// TwinCAT 3 PLC project StudentStation
// ProgramVersion: 3.1.4022.4
// libraries:
//   Tc2_Standard, * (Beckhoff Automation GmbH)
//   Tc2_System, * (Beckhoff Automation GmbH)
//   Tc3_Module, * (Beckhoff Automation GmbH)
//   VisuDialogs, * (System)
//   VisuSymbols,3.5.10.0,System
// project tree:
//   ABBControl/ ABBAssemble.TcPOU, ABBGotoAGVPos.TcPOU, ABBGotoBuffer.TcPOU, ABBGotoHome.TcPOU, ABBGotoScanner.TcPOU, ABBGotoTable.TcPOU, ABBPickLeaveBuffer.TcPOU, ABBPickLeaveContainerAGV.TcPOU, ABBPickLeaveContaineronTable.TcPOU, ABBPickLeaveScanner.TcPOU, ABBScanContainer.TcPOU, ABBScannerStation.TcPOU
//   Automation Library/ AGVControlSystem.TcPOU, AutomationLibrary.TcPOU, BookingSystem.TcPOU, CommData.TcGVL, OrderHandling.TcPOU, PhysicalSystemTest.TcPOU, RobotControlSystem.TcPOU, RobotPosTracker.TcPOU, SensorReader.TcPOU, Visualaisation_Control.TcPOU
//   DUTs/ ABBPositions.TcDUT, ABBXYPOS.TcDUT, OrderPLC.TcDUT, PLCRobotOrder.TcDUT, Station.TcDUT, Storage.TcDUT
//   / GlobalTextList.TcGTLO, PlcTask.TcTTO, Visualization Manager.TcVMO (not stored)
//   GVLs/ GVL.TcGVL
//   POUs/ ABB_Control_FB.TcPOU, MAIN.TcPOU, Scanner_FB.TcPOU, Sensor_Sense.TcPOU
//   VISUs/ RobotStation.TcVIS, Station.TcVIS, Visualization.TcVIS
// real-time tasks:
//   TASK PlcTask: cycle T#10ms, priority 20, ADS port 350

CONFIGURATION StudentStation
    RESOURCE PLC ON TwinCAT3
        TASK PlcTask(INTERVAL := T#10ms, PRIORITY := 20);
        PROGRAM MAIN WITH PlcTask : MAIN;
    END_RESOURCE
END_CONFIGURATION

// ---- DUTs/ABBPositions.TcDUT
TYPE ABBPositions :
STRUCT
	Home: ABBXYPOS;
	Bufferhome: ABBXYPOS;
	Scannerhome: ABBXYPOS;
	Tablehome: ABBXYPOS;
	AGVPOShome: ABBXYPOS;
	Storage1: ABBXYPOS;
	Storage2: ABBXYPOS;
	Storage3: ABBXYPOS;
END_STRUCT
END_TYPE

// ---- DUTs/ABBXYPOS.TcDUT
TYPE ABBXYPOS :
STRUCT
	X:	INT;
	Y:	INT;
END_STRUCT
END_TYPE

// ---- DUTs/OrderPLC.TcDUT
TYPE OrderPLC :
STRUCT
	RobotPOS:STRING; //Prerequest position for the robot to do the step
	PLCorder:INT;	//PLCStep Code
	Robotreply:INT;	//Robot Response Code
END_STRUCT
END_TYPE

// ---- DUTs/PLCRobotOrder.TcDUT
TYPE PLCRobotOrder :
STRUCT
	GotoHome: OrderPLC;
	GotoAGVPos: OrderPLC;
	GotoBuffer: OrderPLC;
	GotoScanner: OrderPLC;
	GotoTable: OrderPLC;
END_STRUCT
END_TYPE

// ---- DUTs/Station.TcDUT
TYPE Station :
STRUCT
	Storage1: Storage;
	Storage2: Storage;
	Storage3: Storage;
END_STRUCT
END_TYPE

// ---- DUTs/Storage.TcDUT
TYPE Storage :
STRUCT
	Component: STRING;
	Quatity: INT;
END_STRUCT
END_TYPE

// ---- Automation Library/CommData.TcGVL
{attribute 'qualified_only'}
VAR_GLOBAL
	msProductNames : ARRAY[1..9] OF STRING := ['BLUECYLINDER', 'BLUEOCTAGON', 'BLUEPLATE', 'YELLOWCYLINDER', 'YELLOWOCTAGON', 'YELLOWPLATE', 'REDCYLINDER', 'REDOCTAGON', 'REDPLATE'];
	mxRequestAGV: BOOL;
	mxAGVOutsideStation: BOOL;
	mxAGVLeaveStation: BOOL;
	mwAGVinStationPOS: INT := -700;
	mwAGVinOutsidePOS: INT := 0;
	mwCurrentAGVPOS: INT;
	ABBPostions: ABBPositions := (Bufferhome := (X := -185, Y := 250), Scannerhome := (X := -185, Y := 180), Tablehome := (X := -185, Y :=350), AGVPOShome := (X := -60, Y := 350), Storage1 := (X := -315, Y := 180), Storage2 := (X := -315, Y := 350), Storage3 := (X := -60, Y := 180));
	mxOnlineMode: BOOL;
	mxABBExecuting: BOOL;
	mwXaxis: INT;
	mwYaxis: INT;
	mxGripper: BOOL;
	mwABBPosXaxis: INT;
	mwABBPosYaxis: INT;
	mxStartABB: BOOL;
	mxScannernoobject:BOOL;
	mxWaitingforSensorinput:BOOL;
	mxNewBookingrequest: BOOL;
	
	
	//Robot Control Signals
	mxRobotOnline AT %I*:BOOL;
	msRobotLastPos:STRING;
	qwOrderRobot AT %Q*:DINT;
	iwReplyRobot AT %I*:DINT;
	qxPLCStrobe AT %Q*:BOOL;
	ixRobotStrobe AT %I*:BOOL;
	iwProgressRobot AT %I*: INT;
	maOrderMaker: ARRAY[1..6] OF INT;
END_VAR

// ---- GVLs/GVL.TcGVL
{attribute 'qualified_only'}
VAR_GLOBAL
	// Order for the next assembly part. The part name should be sent as per the part list and case sensitive. 
	{attribute 'OPC.UA.DA' := '1'}
	qsOrderFornextAssembly AT %Q*: STRING := '0';
	// Parts in your Station buffer. Each buffer have 3 storage locations. The part name and quantity should be mentioned.
	{attribute 'OPC.UA.DA' := '1'}
	BufferProducts AT %Q*: Station;
	// Signal to AGV, a pallet is placed from Station to the AGV. 
	{attribute 'OPC.UA.DA' := '1'}
	qxPalletPlacedinAGV AT %Q*: BOOL;
	// Signal From AGV, that it have docked in your station
	{attribute 'OPC.UA.DA' := '1'}
	ixAGVatStation AT %I*: BOOL;
	{attribute 'OPC.UA.DA' := '1'}	
	qxPickedfromAGV AT %Q*:BOOL; //Part is picked up from the AGV
	{attribute 'OPC.UA.DA' := '1'}
	mwStationStatus AT %Q*: INT; //Pre-Conditioning Mode //100:Ready to Work § 200: Getting Booked § 300: Booked and Busy § 400 : Manual mode  § 500: Pause Mode § 1000 : Emergency Mode 
	{attribute 'OPC.UA.DA' := '1'}	
	// Emergency Stop is active
	ixEmergencyStop AT %Q*:BOOL;
	
	// Inductive sensor reading. from scaning station
	ixInductiveSensor1 AT %I*:BOOL;
	// Inductive sensor reading. from scaning station
	ixInductiveSensor2 AT %I*:BOOL;
	// Inductive sensor reading. from scaning station
	ixInductiveSensor3 AT %I*:BOOL;
	// Inductive sensor reading. from scaning station
	ixInductiveSensor4 AT %I*:BOOL;
	// Inductive sensor reading. from the sensor in robot Tool
	ixInductiveSensorinTool AT %I*:BOOL;
	// Station ID of the station you are working with.
	{attribute 'OPC.UA.DA' := '1'}
	mwStationID AT %Q*: INT;
	
END_VAR

// ---- POUs/MAIN.TcPOU
PROGRAM MAIN
VAR	
END_VAR

VAR_INPUT
	qxABBonlineLamp : BOOL;
	qxABBExecutLamp : BOOL;
	qxABBErrorLamp : BOOL;
	qxPauseLamp : BOOL;
	qxEmergySTLamp : BOOL;
	ixPauseButt : BOOL;
	ixResetABB : BOOL;
	qxAutoMode : BOOL;
	qxManualMode : BOOL;
	ixAutoLamp : BOOL;
	ixManualLamp : BOOL;
	qxDoneContainerScan : BOOL;
	qxDoneBuffer1Scan : BOOL;
	qsContainer : STRING;
	qsTask : STRING;
	qsSubTask : STRING;
	mxPlateAvailable : BOOL;
	mxCylinderAvailable : BOOL;
	mxOctagonAvailable : BOOL;
	mwBufferID : INT;
	ixEmptyBuffer : BOOL;
	mwPartID : INT;
	sPartID : ARRAY [1..3] OF STRING:= ['Part 1', 'Part 2', 'Part 3'];
END_VAR

VAR_OUTPUT
	
END_VAR

AutomationLibrary();
Visualaisation_Control();
RobotPosTracker();
ABB_Control_FB();

END_PROGRAM

// ---- Automation Library/AutomationLibrary.TcPOU
PROGRAM AutomationLibrary
VAR
	OrderHandling_Global: OrderHandling;
	mxErrorCodeOrder: INT;
	AGVControlSystem_GLobal: AGVControlSystem;
	RobotControlSystem_Global: RobotControlSystem;
	ABBGotoHome_TEST: ABBGotoHome;
	mxEnable: BOOL;
	BookingSystem_Global: BookingSystem;
	mxBookingDone: BOOL;
	mxBookingError: BOOL;
END_VAR

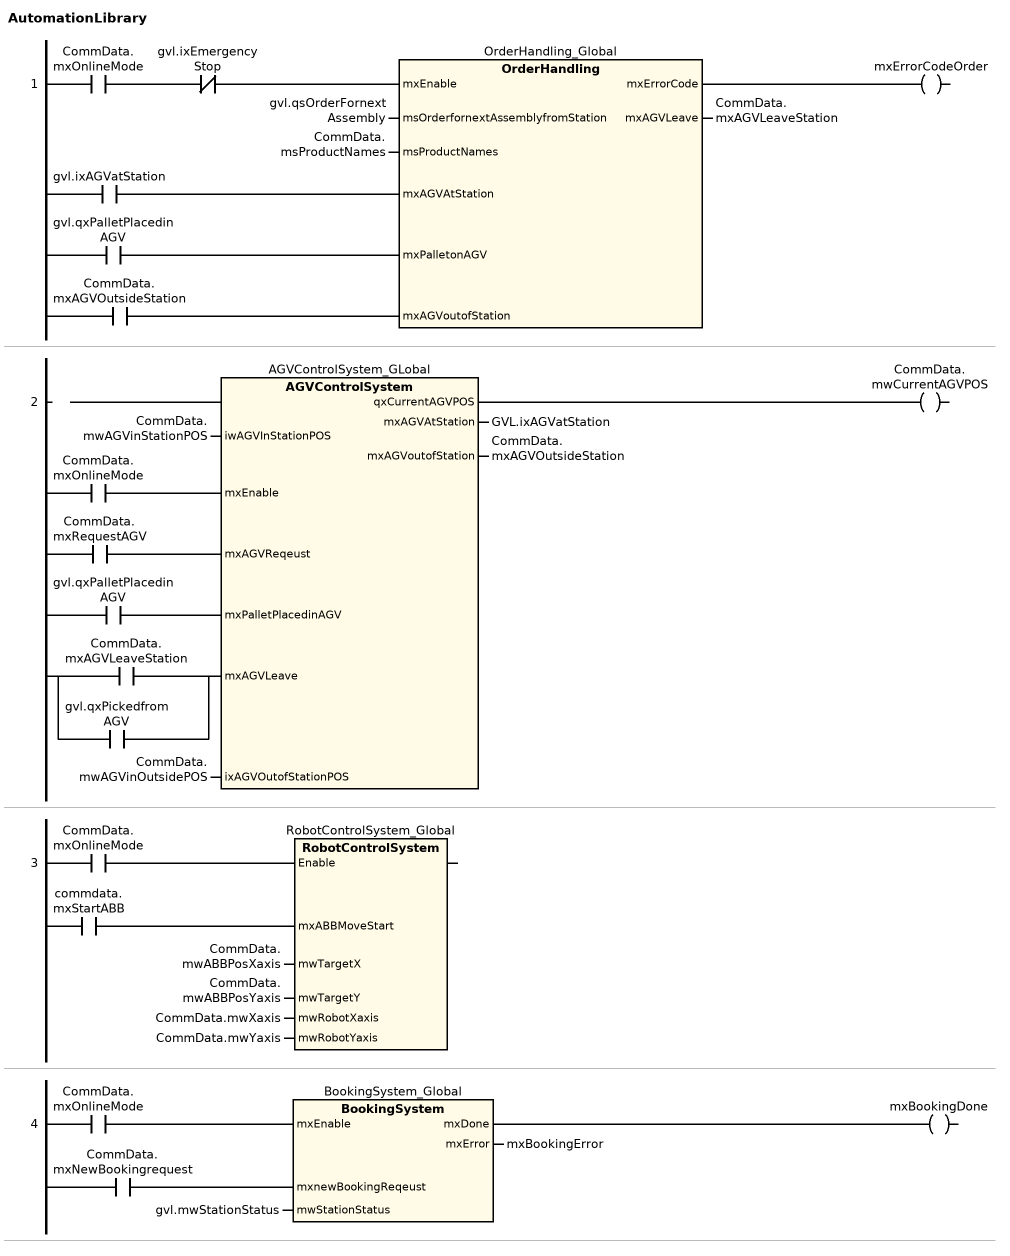
// NETWORK 1
OrderHandling_Global(
    mxEnable := CommData.mxOnlineMode AND NOT gvl.ixEmergencyStop,
    msOrderfornextAssemblyfromStation := gvl.qsOrderFornextAssembly,
    msProductNames := CommData.msProductNames,
    mxAGVAtStation := gvl.ixAGVatStation,
    mxPalletonAGV := gvl.qxPalletPlacedinAGV,
    mxAGVoutofStation := CommData.mxAGVOutsideStation,
    mxAGVLeave => CommData.mxAGVLeaveStation); // OrderHandling
mxErrorCodeOrder := OrderHandling_Global.mxErrorCode;

// NETWORK 2
AGVControlSystem_GLobal(
    iwAGVInStationPOS := CommData.mwAGVinStationPOS,
    mxEnable := CommData.mxOnlineMode,
    mxAGVReqeust := CommData.mxRequestAGV,
    mxPalletPlacedinAGV := gvl.qxPalletPlacedinAGV,
    mxAGVLeave := CommData.mxAGVLeaveStation OR gvl.qxPickedfromAGV,
    ixAGVOutofStationPOS := CommData.mwAGVinOutsidePOS,
    mxAGVAtStation => GVL.ixAGVatStation,
    mxAGVoutofStation => CommData.mxAGVOutsideStation); // AGVControlSystem
CommData.mwCurrentAGVPOS := AGVControlSystem_GLobal.qxCurrentAGVPOS;

// NETWORK 3
RobotControlSystem_Global(
    Enable := CommData.mxOnlineMode,
    mxABBMoveStart := commdata.mxStartABB,
    mwTargetX := CommData.mwABBPosXaxis,
    mwTargetY := CommData.mwABBPosYaxis,
    mwRobotXaxis := CommData.mwXaxis,
    mwRobotYaxis := CommData.mwYaxis); // RobotControlSystem

// NETWORK 4
BookingSystem_Global(
    mxEnable := CommData.mxOnlineMode,
    mxnewBookingReqeust := CommData.mxNewBookingrequest,
    mwStationStatus := gvl.mwStationStatus,
    mxError => mxBookingError); // BookingSystem
mxBookingDone := BookingSystem_Global.mxDone;

END_PROGRAM

// ---- Automation Library/OrderHandling.TcPOU
FUNCTION_BLOCK OrderHandling
VAR_INPUT
	mxEnable: BOOL;
	msOrderfornextAssemblyfromStation: STRING;
	msProductNames: Array[1..9] OF STRING;
	mxAGVAtStation: BOOL;
	mxPalletonAGV: BOOL;
	mxAGVoutofStation: BOOL;
END_VAR
VAR_OUTPUT
	mxErrorCode: INT;
	mxAGVLeave: BOOL;
END_VAR
VAR
	order: INT;
END_VAR

IF mxEnable THEN
	CASE order OF
		0:
			IF msOrderfornextAssemblyfromStation <> '0' THEN
				order:= 10;
			END_IF
		10:
			order:=20;
		20:
			IF msOrderfornextAssemblyfromStation = msProductNames[1] THEN
				order:=30;
			ELSIF msOrderfornextAssemblyfromStation = msProductNames[2] THEN
				order:=30;
			ELSIF msOrderfornextAssemblyfromStation = msProductNames[3] THEN
				order:=30;
			ELSIF msOrderfornextAssemblyfromStation = msProductNames[4] THEN
				order:=30;
			ELSIF msOrderfornextAssemblyfromStation = msProductNames[5] THEN
				order:=30;
			ELSIF msOrderfornextAssemblyfromStation = msProductNames[6] THEN
				order:=30;
			ELSIF msOrderfornextAssemblyfromStation = msProductNames[7] THEN
				order:=30;
			ELSIF msOrderfornextAssemblyfromStation = msProductNames[8] THEN
				order:=30;
			ELSIF msOrderfornextAssemblyfromStation = msProductNames[9] THEN
				order:=30;
			ELSIF msOrderfornextAssemblyfromStation = 'AssembledProduct' THEN
				order:=30;
			ELSIF msOrderfornextAssemblyfromStation = 'InvalidPart' THEN
				order:=30;
			ELSE 
				order:=22;
			END_IF 
		22: // Invalid Product Name
			mxErrorCode:=22;
				IF msOrderfornextAssemblyfromStation = '0' THEN
					mxErrorCode:=0;
					order:= 0;
				END_IF
		30:
			CommData.mxRequestAGV:=TRUE;
			IF mxAGVAtStation THEN
				CommData.mxRequestAGV:=FALSE;
				order:=40;
			END_IF
		40:
			IF mxPalletonAGV THEN
				mxAGVLeave:=TRUE;
				order:=50;
			END_IF
		50:
			IF mxAGVoutofStation THEN
				mxAGVLeave:=FALSE;
				order:=60;
			END_IF
		60:
			IF msOrderfornextAssemblyfromStation = '0' THEN
				order:= 0;
			END_IF
	END_CASE
END_IF

END_FUNCTION_BLOCK

// ---- Automation Library/AGVControlSystem.TcPOU
FUNCTION_BLOCK AGVControlSystem
VAR
	AGV: INT;
	mxAGVMoveTarget: INT;
	iwAGVOutofStationPOS: INT;
	RSpeed:INT:=1;
END_VAR
VAR_INPUT
	iwAGVInStationPOS: INT;
	mxEnable: BOOL;
END_VAR
VAR_OUTPUT
	qxCurrentAGVPOS: INT := 0;
	mxAGVAtStation: BOOL;
	mxAGVoutofStation: BOOL;
END_VAR
VAR_INPUT
	mxAGVReqeust: BOOL;
	mxPalletPlacedinAGV: BOOL;
	mxAGVLeave: BOOL;
	ixAGVOutofStationPOS: INT;
END_VAR

IF mxEnable THEN
	
	CASE AGV OF
		0:
			IF mxAGVReqeust THEN
				AGV:=10;
			END_IF
		10:
			mxAGVMoveTarget:= iwAGVInStationPOS;
			AGV:=20;
		20:
			
			IF mxAGVMoveTarget < qxCurrentAGVPOS THEN
				qxCurrentAGVPOS:=qxCurrentAGVPOS-RSpeed;
				AGV:=30;
			END_IF
		30:
			IF mxAGVMoveTarget < qxCurrentAGVPOS THEN
				AGV:=20;
			ELSIF  mxAGVMoveTarget >= qxCurrentAGVPOS THEN
				AGV:=40;
			END_IF
		40:
			mxAGVAtStation:=TRUE;
			IF mxPalletPlacedinAGV OR mxAGVLeave THEN
				mxAGVAtStation:=FALSE;
				AGV:=50;
			END_IF
		50:
			mxAGVMoveTarget:= iwAGVOutofStationPOS;
			AGV:=60;
		60:
			IF mxAGVMoveTarget > qxCurrentAGVPOS THEN
				qxCurrentAGVPOS:=qxCurrentAGVPOS+RSpeed;
				AGV:=70;
			END_IF
		70:
			IF mxAGVMoveTarget > qxCurrentAGVPOS THEN
				AGV:=60;
			ELSIF  mxAGVMoveTarget <= qxCurrentAGVPOS THEN
				AGV:=80;
			END_IF
		80:
			mxAGVoutofStation:=TRUE;
			IF NOT mxAGVReqeust AND NOT mxAGVLeave THEN
				mxAGVoutofStation:=FALSE;
				AGV:=0;
			END_IF
	END_CASE
		
END_IF

END_FUNCTION_BLOCK

// ---- Automation Library/RobotControlSystem.TcPOU
FUNCTION_BLOCK RobotControlSystem
VAR_INPUT
	Enable: BOOL;
	mxABBMoveStart: BOOL;
	mwTargetX: INT;
	mwTargetY: INT;
END_VAR
VAR_OUTPUT
END_VAR
VAR
	ABBMove: INT;
	RSpeed:INT:=1;
END_VAR

VAR_IN_OUT
	mwRobotXaxis: INT;
	mwRobotYaxis: INT;
END_VAR

IF Enable THEN
	CASE ABBMove OF
		0:
			IF mxABBMoveStart THEN
				ABBMove:=10;
			END_IF
		10:
			IF NOT CommData.mxABBExecuting THEN
				CommData.mxABBExecuting:=TRUE;
				ABBMove:=20;
			END_IF
		20:
			IF mwRobotXaxis < mwTargetX THEN
				mwRobotXaxis :=mwRobotXaxis+RSpeed;
				ABBMove:=30;
			ELSIF mwRobotXaxis > mwTargetX THEN
				mwRobotXaxis :=mwRobotXaxis-RSpeed;
				ABBMove:=30;
			ELSIF mwRobotXaxis = mwTargetX THEN
				ABBMove:=30;
			END_IF
		30:
			IF mwRobotYaxis < mwTargetY THEN
				mwRobotYaxis :=mwRobotYaxis+RSpeed;
				ABBMove:=40;
			ELSIF mwRobotYaxis > mwTargetY THEN
				mwRobotYaxis :=mwRobotYaxis-RSpeed;
				ABBMove:=40;
			ELSIF mwRobotYaxis = mwTargetY THEN
				ABBMove:=40;
			END_IF
		40:
			IF mwRobotXaxis = mwTargetX AND mwRobotYaxis = mwTargetY THEN
				ABBMove:=50;
			ELSIF gvl.ixEmergencyStop THEN
				ABBMove:=50;
			ELSE
				ABBMOve:=20;
			END_IF
		50:
			CommData.mxABBExecuting:=FALSE;
			IF NOT mxABBMoveStart THEN
				ABBMove:=0;
			END_IF
	END_CASE
END_IF

END_FUNCTION_BLOCK

// ---- ABBControl/ABBGotoHome.TcPOU
FUNCTION_BLOCK ABBGotoHome
VAR_INPUT
	mxEnable: BOOL;
END_VAR
VAR_OUTPUT
	mxDone:BOOL;
	mxExecuting: BOOL;
	mxError: BOOL;
END_VAR
VAR
	ABB: INT;
END_VAR

CASE ABB OF
	0:
		IF mxEnable AND NOT CommData.mxABBExecuting THEN
			ABB:=10;
		END_IF
	10:
		IF CommData.mxRobotOnline THEN
			ABB:=100;
			ELSE
			ABB:=200;
		END_IF
	100:
		mxExecuting:=TRUE;
		CommData.maOrderMaker[1] := 1;
		CommData.maOrderMaker[2] := 0;
		CommData.maOrderMaker[3] := 0;
		CommData.maOrderMaker[4] := 0;
		CommData.maOrderMaker[5] := 0;
		CommData.maOrderMaker[6] := 0;
		CommData.qwOrderRobot:=100000;
		ABB:=101;
	101:
		IF CommData.qwOrderRobot > 0 THEN
			CommData.qxPLCStrobe:=TRUE;
			ABB:=102;
		END_IF
	102:
		IF CommData.ixRobotStrobe THEN
			IF CommData.iwReplyRobot = CommData.qwOrderRobot+1 THEN
				CommData.qwOrderRobot:=0;
				CommData.maOrderMaker[1] := 0;
				CommData.maOrderMaker[2] := 0;
				CommData.maOrderMaker[3] := 0;
				CommData.maOrderMaker[4] := 0;
				CommData.maOrderMaker[5] := 0;
				CommData.maOrderMaker[6] := 0;
				CommData.qxPLCStrobe:=FALSE;
				ABB:=103;
			ELSE
				ABB:=1000;
			END_IF
		END_IF
	103:
		IF NOT CommData.ixRobotStrobe THEN
			IF CommData.iwReplyRobot = 0 THEN
				ABB:=104;
			ELSE
				ABB:=1000;
			END_IF
		END_IF
	104:
		IF CommData.ixRobotStrobe THEN
			IF CommData.iwProgressRobot = 90 THEN
				CommData.qxPLCStrobe:=TRUE;
				ABB:=105;
			END_IF
			IF CommData.iwProgressRobot = 1000 THEN
				CommData.qxPLCStrobe:=TRUE;
				ABB:=1000;
			END_IF
		END_IF	
	105:
		IF  NOT CommData.ixRobotStrobe AND CommData.iwProgressRobot = 0 THEN
			CommData.qxPLCStrobe:=FALSE;
			ABB:=201;
		END_IF
	
	200:
		CommData.mwABBPosXaxis:=CommData.ABBPostions.Home.X;
		CommData.mwABBPosYaxis:=CommData.ABBPostions.Home.Y;
		mxExecuting:=TRUE;
		CommData.mxStartABB:=TRUE;
		IF CommData.mwXaxis = CommData.ABBPostions.Home.X AND CommData.mwYaxis = CommData.ABBPostions.Home.Y THEN
			ABB:=201;
		ELSIF gvl.ixEmergencyStop THEN
			ABB:=1000;
		END_IF
	201:
		mxExecuting:=FALSE;
		CommData.mxStartABB:=FALSE;
		mxDone:=TRUE;
		IF NOT mxEnable THEN
			mxDone:=FALSE;
			ABB:=0;
		END_IF
	1000:
		mxError:=TRUE;
		mxExecuting:=FALSE;
		CommData.mxStartABB:=FALSE;
		IF NOT mxEnable THEN
			mxError:=FALSE;
			mxDone:=FALSE;
			ABB:=0;
		END_IF
END_CASE



IF gvl.ixEmergencyStop THEN
	ABB:=1000;
END_IF

END_FUNCTION_BLOCK

// ---- Automation Library/BookingSystem.TcPOU
FUNCTION_BLOCK BookingSystem
VAR_INPUT
	mxEnable: BOOL;
	mxnewBookingReqeust: BOOL;
END_VAR
VAR_OUTPUT
	mxDone:BOOL;
	mxError:BOOL;
END_VAR
VAR
	booking: INT;
END_VAR

VAR_IN_OUT
	mwStationStatus: INT;
END_VAR

IF mxEnable THEN
	CASE booking OF
		0:
		 	IF mxnewBookingReqeust THEN
				booking:=10;
			END_IF
		10:
			IF mwStationStatus =100 THEN
				booking:=20;
			ELSE 
				booking:=1000;
			END_IF
		20:
			mwStationStatus:=200;
			booking:=30;
		30:
			mxDone:=TRUE;
			IF NOT mxnewBookingReqeust THEN
				mxDone:=FALSE;
				booking:=0;
			END_IF
		1000:
			mxError:=TRUE;
			IF NOT mxnewBookingReqeust THEN
				mxDone:=FALSE;
				mxError:=FALSE;
				booking:=0;
			END_IF
	END_CASE
END_IF

END_FUNCTION_BLOCK

// ---- Automation Library/Visualaisation_Control.TcPOU
PROGRAM Visualaisation_Control
VAR
	mxDebugButton: BOOL;
	mxDebugMode: BOOL;
	mxStationStatus: STRING;
	mxManualMode: BOOL;
END_VAR

IF mxDebugButton THEN
	mxDebugMode:=TRUE;
ELSE
	mxDebugMode:=FALSE;
END_IF

//100:Ready to Work § 200: Getting Booked § 300: Booked and Busy § 400 : Manual mode  § 500: Pause Mode § 1000 : Emergency Mode 
IF gvl.mwStationStatus = 100 THEN
	mxStationStatus:= 'Ready for Order';
	mxManualMode:=FALSE;
ELSIF gvl.mwStationStatus = 200 THEN
	mxStationStatus:= 'Executing booking order from IOStation';
	mxManualMode:=FALSE;
ELSIF gvl.mwStationStatus = 300 THEN
	mxStationStatus:= 'Booked for Order or Busy';
	mxManualMode:=FALSE;
ELSIF gvl.mwStationStatus = 400 THEN
	mxStationStatus:= 'Manual Mode';
	mxManualMode:=TRUE;
ELSIF gvl.mwStationStatus = 500 THEN
	mxStationStatus:= 'Pause Mode';
ELSIF gvl.mwStationStatus = 1000 OR  gvl.ixEmergencyStop THEN
	mxStationStatus:= 'Emergency Mode';
	mxManualMode:=FALSE;
ELSIF gvl.mwStationStatus = 0 THEN
	mxStationStatus:= 'Intial Mode';
	mxManualMode:=FALSE;
ELSIF  gvl.mwStationStatus = 50 THEN
	mxStationStatus:= 'Pre-Condition State';
ELSE
	mxStationStatus:= 'Status Unknown';
END_IF

END_PROGRAM

// ---- Automation Library/RobotPosTracker.TcPOU
PROGRAM RobotPosTracker
VAR
	Robot: INT;
	maLastOrder:ARRAY[1..6] OF INT;
END_VAR

CASE Robot OF
	0:
		IF CommData.mxRobotOnline THEN
			Robot:=10;
		END_IF
	10:
		IF CommData.qxPLCStrobe THEN
			maLastOrder:=CommData.maOrderMaker;
			Robot:=20;
		END_IF
	20:
		IF CommData.iwProgressRobot =90 AND CommData.ixRobotStrobe THEN
			Robot:=30;
		END_IF
	30:
		IF maLastOrder[1] = 1 THEN
			IF maLastOrder[6] = 0 THEN
				Robot:=40;
			ELSIF maLastOrder[6] = 5 THEN
				Robot:=41;
			END_IF
		ELSIF  maLastOrder[1] = 2 THEN
			IF maLastOrder[6] = 0 THEN
				Robot:=42;
			ELSIF maLastOrder[6] = 5 THEN
				Robot:=43;
			END_IF
		ELSIF  maLastOrder[1] = 3 THEN
			Robot:=44;
		ELSIF maLastOrder[1] = 4 THEN
			Robot:=45;
		ELSIF maLastOrder[1] = 5 THEN
			Robot:=46;
		ELSIF maLastOrder[1] = 6 THEN
			Robot:=47;
		ELSIF maLastOrder[1] = 7 THEN
			Robot:=48;
		ELSIF maLastOrder[1] = 8 THEN
			Robot:=49;
		ELSIF maLastOrder[1] = 9 THEN
			Robot:=50;
		END_IF 
	40:
		CommData.msRobotLastPos:='Home';
		Robot:=1000;
	41:
		CommData.msRobotLastPos:='Buffer';
		Robot:=1000;
	42:
		CommData.msRobotLastPos:='AGV';
		Robot:=1000;
	43:
		CommData.msRobotLastPos:='Scanner';
		Robot:=1000;
	44:
		CommData.msRobotLastPos:='Table';
		Robot:=1000;
		
	45:
		CommData.msRobotLastPos:='AGV';
		Robot:=1000;
	46:
		CommData.msRobotLastPos:='Table';
		Robot:=1000;
	47:
		CommData.msRobotLastPos:='Scanner';
		Robot:=1000;
	48:
		CommData.msRobotLastPos:='Table';
		Robot:=1000;
	49:
		CommData.msRobotLastPos:='Table';
		Robot:=1000;
	50:
		CommData.msRobotLastPos:='Buffer';
		Robot:=1000;
		
	1000:
		IF CommData.iwProgressRobot =0 AND NOT CommData.qxPLCStrobe THEN
			Robot:=0;
		END_IF
END_CASE

END_PROGRAM

// ---- POUs/ABB_Control_FB.TcPOU
PROGRAM ABB_Control_FB
VAR_INPUT
	mxScan: BOOL;
	qxCon1: BOOL;
	mxCon_1_ATtableScan: BOOL;
	qxCon2: BOOL;
	mxCon_2_ATtableScan: BOOL;
	qxCon3: BOOL;
	mxCon_3_ATtableScan: BOOL;
	qxPart_1_Assemble: BOOL;
	qxPart_2_Assemble: BOOL;
	qxPart_3_Assemble: BOOL;
	ixGoTo_AGV: BOOL;
	qxScanBuffer_1: BOOL;
	qxScanBuffer_2: BOOL;
	qxScanBuffer_3: BOOL;
	qxAssemblyDone: BOOL;
	mxConLeave: BOOL;
	qxGotoHome: BOOL;
	ixGotoHome: BOOL;
	qxGotoTable: BOOL;
	ixGotoTable: BOOL;
	qxGotoAGV: BOOL;
	ixGotoAGV: BOOL;
	qxGotoScanner: BOOL;
	ixGotoScanner: BOOL;
	qxGotoBuffer: BOOL;
	ixGotoBuffer: BOOL;
	qxPickBuffer1: BOOL;
	ixPickBuffer1: BOOL;
	qxPickBuffer2: BOOL;
	ixPickBuffer2: BOOL;
	qxPickBuffer3: BOOL;
	ixPickBuffer3: BOOL;
	qxLeaveBuffer1: BOOL;
	ixLeaveBuffer1: BOOL;
	qxLeaveBuffer2: BOOL;
	ixLeaveBuffer2: BOOL;
	qxLeaveBuffer3: BOOL;
	ixLeaveBuffer3: BOOL;
	qxPickScanner: BOOL;
	ixPickScanner: BOOL;
	qxLeaveScanner: BOOL;
	ixLeaveScanner: BOOL;
	qxPickAGV: BOOL;
	ixPickAGV: BOOL;
	qxLeaveAGV: BOOL;
	ixLeaveAGV: BOOL;
	qxPickTable: BOOL;
	ixPickTable: BOOL;
	qxLeaveTable: BOOL;
	ixLeaveTable: BOOL;
	ixScanBuffer: BOOL;
	ixScanContainer: BOOL;
	ixScanPart1: BOOL;
	ixScanPart2: BOOL;
	ixScanPart3: BOOL;
	ixAssemble1: BOOL;
	ixAssemble2: BOOL;
	ixAssemble3: BOOL;
	ixSendOrder: BOOL;
	ixFinishOrder: BOOL;
	mxAsse_1_done: BOOL;
	mxAsse_2_done: BOOL;
	mxAsse_3_done: BOOL;
END_VAR

VAR
	ABBGotoHome_1: ABBGotoHome;
	Auto_Mode: RS;
	Manual_Mode: RS;
	ABBGotoBufferPick_1: ABBGotoBuffer;
	ABBPickLeaveBufferPick_1: ABBPickLeaveBuffer;
	ABBGotoScanner_1: ABBGotoScanner;
	ABBPickLeaveScannerLB_1: ABBPickLeaveScanner;
	SensorReader_buffer_1: SensorReader;
	ABBScannerStation_1: ABBScannerStation;
	ABBPickLeaveScannerPB_1: ABBPickLeaveScanner;
	ABBGotoBufferLeave_1: ABBGotoBuffer;
	ABBPickLeaveBufferLeave_1: ABBPickLeaveBuffer;
	mxBuffer_1_scanned: BOOL;
	Reading_1_Done: RS;
	ABBGotoBufferPick_2: ABBGotoBuffer;
	ABBPickLeaveBufferPick_2: ABBPickLeaveBuffer;
	ABBGotoScanner_2: ABBGotoScanner;
	ABBPickLeaveScannerLB_2: ABBPickLeaveScanner;
	ABBScannerStation_2: ABBScannerStation;
	ABBPickLeaveScannerPB_2: ABBPickLeaveScanner;
	ABBGotoBufferLeave_2: ABBGotoBuffer;
	ABBPickLeaveBufferLeave_2: ABBPickLeaveBuffer;
	mxBuffer_2_scanned: BOOL;
	ABBGotoBufferPick_3: ABBGotoBuffer;
	ABBPickLeaveBufferPick_3: ABBPickLeaveBuffer;
	ABBGotoScanner_3: ABBGotoScanner;
	ABBPickLeaveScannerLB_3: ABBPickLeaveScanner;
	ABBScannerStation_3: ABBScannerStation;
	ABBPickLeaveScannerPB_3: ABBPickLeaveScanner;
	ABBGotoBufferLeave_3: ABBGotoBuffer;
	ABBPickLeaveBufferLeave_3: ABBPickLeaveBuffer;
	mxBuffer_3_scanned: BOOL;
	ABBGotoHome_AGV_Con1: ABBGotoHome;
	SensorReader_0: SensorReader;
	Scanner_FB_0: Scanner_FB;
	mxRP: BOOL;
	mxYP: BOOL;
	mxBP: BOOL;
	mxRCy: BOOL;
	mxYCy: BOOL;
	mxBCy: BOOL;
	mxYOct: BOOL;
	mxBOct: BOOL;
	mxROct: BOOL;
	mxIP: BOOL;
	Sensor_Sense_0: Sensor_Sense;
	mxRCon: BOOL;
	mxYCon: BOOL;
	mxBCon: BOOL;
	mxContainerScanDone: BOOL;
	mxScanner: BOOL;
	Scan_Block: RS;
	mxScanDone: BOOL;
	ABBGotoAGVPos_1: ABBGotoAGVPos;
	ABBPickLeaveContainerAGV_1: ABBPickLeaveContainerAGV;
	ABBGotoScannerCon_1: ABBGotoScanner;
	ABBPickLeaveContainerAGVPick_1: ABBPickLeaveContainerAGV;
	ABBPickLeaveContainerAGVLeave_1: ABBPickLeaveContainerAGV;
	ABBPickLeaveScannerLC_1: ABBPickLeaveScanner;
	ABBScanContainer_1: ABBScanContainer;
	ABBScannerStationCon1_1: ABBScannerStation;
	ABBPickLeaveScannerPC_1: ABBPickLeaveScanner;
	ABBGotoTableCon_1: ABBGotoTable;
	ABBGotoTableCon_1_Scanned: ABBGotoTable;
	ABBGotoTableCon_2: ABBGotoTable;
	ABBScanContainer_2: ABBScanContainer;
	ABBGotoTableCon_2_Scanned: ABBGotoTable;
	ABBGotoTableCon_3: ABBGotoTable;
	ABBScanContainer_3: ABBScanContainer;
	ABBGotoTableCon_3_Scanned: ABBGotoTable;
	ABBAssemble_1: ABBAssemble;
	ABBGotoTable_Ass1: ABBGotoTable;
	
	ABBAssemble_2: ABBAssemble;
	ABBGotoTable_Ass2: ABBGotoTable;
	
	ABBAssemble_3: ABBAssemble;
	ABBGotoTable_Ass3: ABBGotoTable;
	
	TON_0: TON;
	ABBPickLeaveContaineronTableLeave_1: ABBPickLeaveContaineronTable;
	ABBPickLeaveContaineronTableLeave_2: ABBPickLeaveContaineronTable;
	ABBPickLeaveContaineronTableLeave_3: ABBPickLeaveContaineronTable;
	ABBGotoTable_0: ABBGotoTable;
	ABBPickLeaveContaineronTableLeave_0: ABBPickLeaveContaineronTable;
	TON_1: TON;
	TON_2: TON;
	TON_3: TON;
	ABBGotoTable_Assembled: ABBGotoTable;
	ABBPickLeaveContaineronTable_Assembled: ABBPickLeaveContaineronTable;
	ABBGotoAGVPos_Assembled: ABBGotoAGVPos;
	ABBPickLeaveContainerAGV_Assembled: ABBPickLeaveContainerAGV;
	ABBAssemble_Part1: ABBAssemble;
	ABBAssemble_Part2: ABBAssemble;
	ABBAssemble_Part3: ABBAssemble;
	ABBGotoHome_Next_Assemnbly: ABBGotoHome;
	mxWaitforNext: BOOL;
	ABBGotoHome_10: ABBGotoHome;
	qxHOME: BOOL;
	ABBGotoTable_10: ABBGotoTable;
	qxTABLE: BOOL;
	ABBGotoAGVPos_10: ABBGotoAGVPos;
	qxAGV: BOOL;
	ABBGotoScanner_10: ABBGotoScanner;
	qxSCANNER: BOOL;
	ABBGotoBuffer_10: ABBGotoBuffer;
	qxBUFFER: BOOL;
	ABBPickLeaveBuffer_Pick: ABBPickLeaveBuffer;
	qxBufferPicked1: BOOL;
	ABBPickLeaveBuffer_Leave: ABBPickLeaveBuffer;
	qxBufferLeft1: BOOL;
	ABBGotoScanner_Pick: ABBGotoScanner;
	ABBPickLeaveScanner_Pick: ABBPickLeaveScanner;
	qxPickedScanner: BOOL;
	ABBGotoScanner_Leave: ABBGotoScanner;
	ABBPickLeaveScanner_Leave: ABBPickLeaveScanner;
	qxLeftScanner: BOOL;
	ABBGotoAGVPos_Pick: ABBGotoAGVPos;
	ABBPickLeaveContainerAGV_Pick: ABBPickLeaveContainerAGV;
	qxPickedAGV: BOOL;
	ABBGotoAGVPos_Leave: ABBGotoAGVPos;
	ABBPickLeaveContainerAGV_Leave: ABBPickLeaveContainerAGV;
	qxLeftAGV: BOOL;
	ABBGotoTable_Pick: ABBGotoTable;
	ABBPickLeaveContaineronTable_Pick: ABBPickLeaveContaineronTable;
	qxPickedTable: BOOL;
	ABBGotoTable_Leave: ABBGotoTable;
	ABBPickLeaveContaineronTable_Leave: ABBPickLeaveContaineronTable;
	qxLeftTable: BOOL;
END_VAR
VAR // added by the converter: edge detectors and wires of the graphical bodies
    _w1, _w2, _w3, _w4, _w5, _w6, _w7 : BOOL;
END_VAR

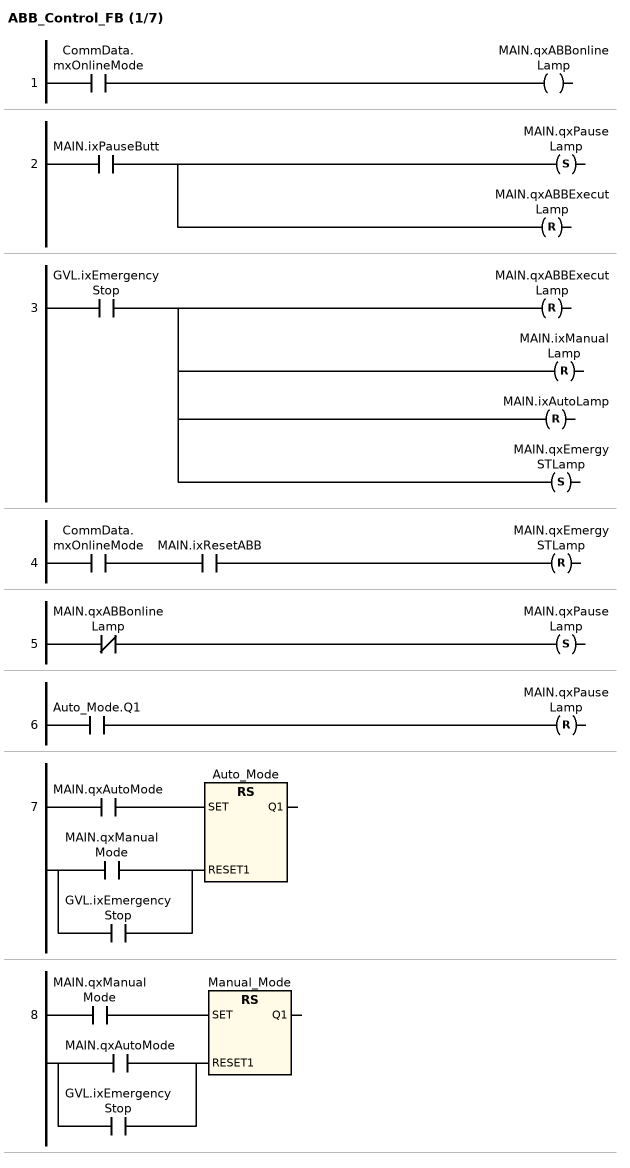
// NETWORK 1
MAIN.qxABBonlineLamp := CommData.mxOnlineMode;

// NETWORK 2
_w1 := MAIN.ixPauseButt;
MAIN.qxPauseLamp S= _w1;
MAIN.qxABBExecutLamp R= _w1;

// NETWORK 3
MAIN.qxABBExecutLamp R= GVL.ixEmergencyStop;
MAIN.ixManualLamp R= GVL.ixEmergencyStop;
MAIN.ixAutoLamp R= GVL.ixEmergencyStop;
MAIN.qxEmergySTLamp S= GVL.ixEmergencyStop;

// NETWORK 4
MAIN.qxEmergySTLamp R= CommData.mxOnlineMode AND MAIN.ixResetABB;

// NETWORK 5
MAIN.qxPauseLamp S= NOT MAIN.qxABBonlineLamp;

// NETWORK 6
MAIN.qxPauseLamp R= Auto_Mode.Q1;

// NETWORK 7
Auto_Mode(SET := MAIN.qxAutoMode, RESET1 := MAIN.qxManualMode OR GVL.ixEmergencyStop); // RS

// NETWORK 8
Manual_Mode(SET := MAIN.qxManualMode, RESET1 := MAIN.qxAutoMode OR GVL.ixEmergencyStop); // RS

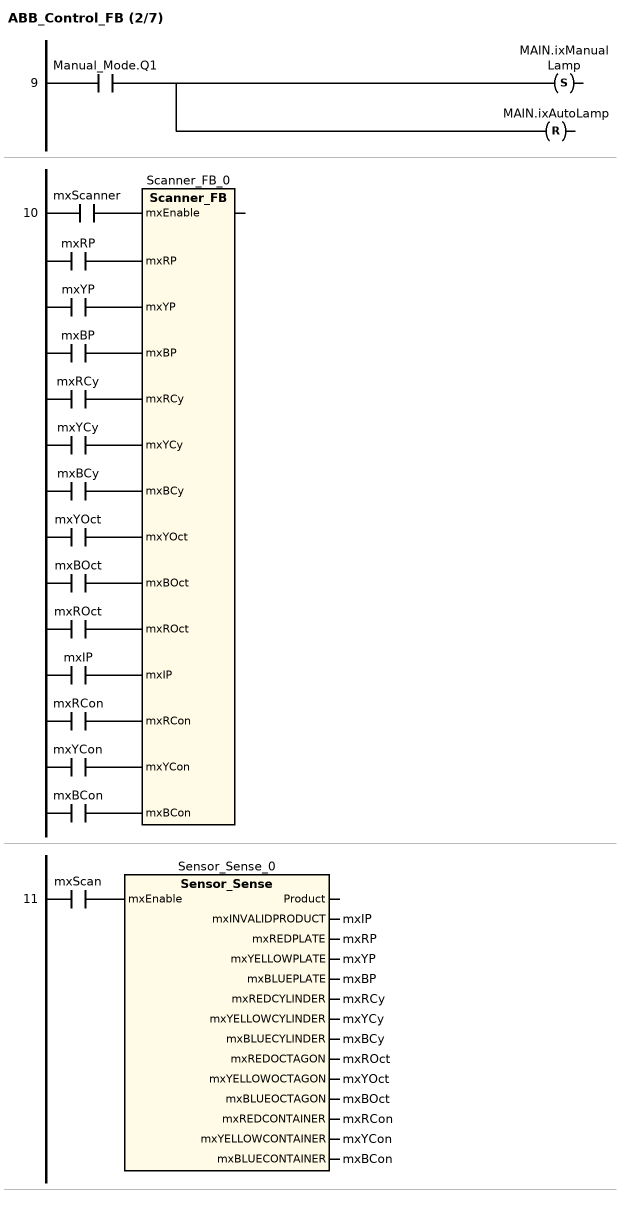
// NETWORK 9
MAIN.ixManualLamp S= Manual_Mode.Q1;
MAIN.ixAutoLamp R= Manual_Mode.Q1;

// NETWORK 10
Scanner_FB_0(
    mxEnable := mxScanner,
    mxRP := mxRP,
    mxYP := mxYP,
    mxBP := mxBP,
    mxRCy := mxRCy,
    mxYCy := mxYCy,
    mxBCy := mxBCy,
    mxYOct := mxYOct,
    mxBOct := mxBOct,
    mxROct := mxROct,
    mxIP := mxIP,
    mxRCon := mxRCon,
    mxYCon := mxYCon,
    mxBCon := mxBCon); // Scanner_FB

// NETWORK 11
Sensor_Sense_0(
    mxEnable := mxScan,
    mxINVALIDPRODUCT => mxIP,
    mxREDPLATE => mxRP,
    mxYELLOWPLATE => mxYP,
    mxBLUEPLATE => mxBP,
    mxREDCYLINDER => mxRCy,
    mxYELLOWCYLINDER => mxYCy,
    mxBLUECYLINDER => mxBCy,
    mxREDOCTAGON => mxROct,
    mxYELLOWOCTAGON => mxYOct,
    mxBLUEOCTAGON => mxBOct,
    mxREDCONTAINER => mxRCon,
    mxYELLOWCONTAINER => mxYCon,
    mxBLUECONTAINER => mxBCon); // Sensor_Sense

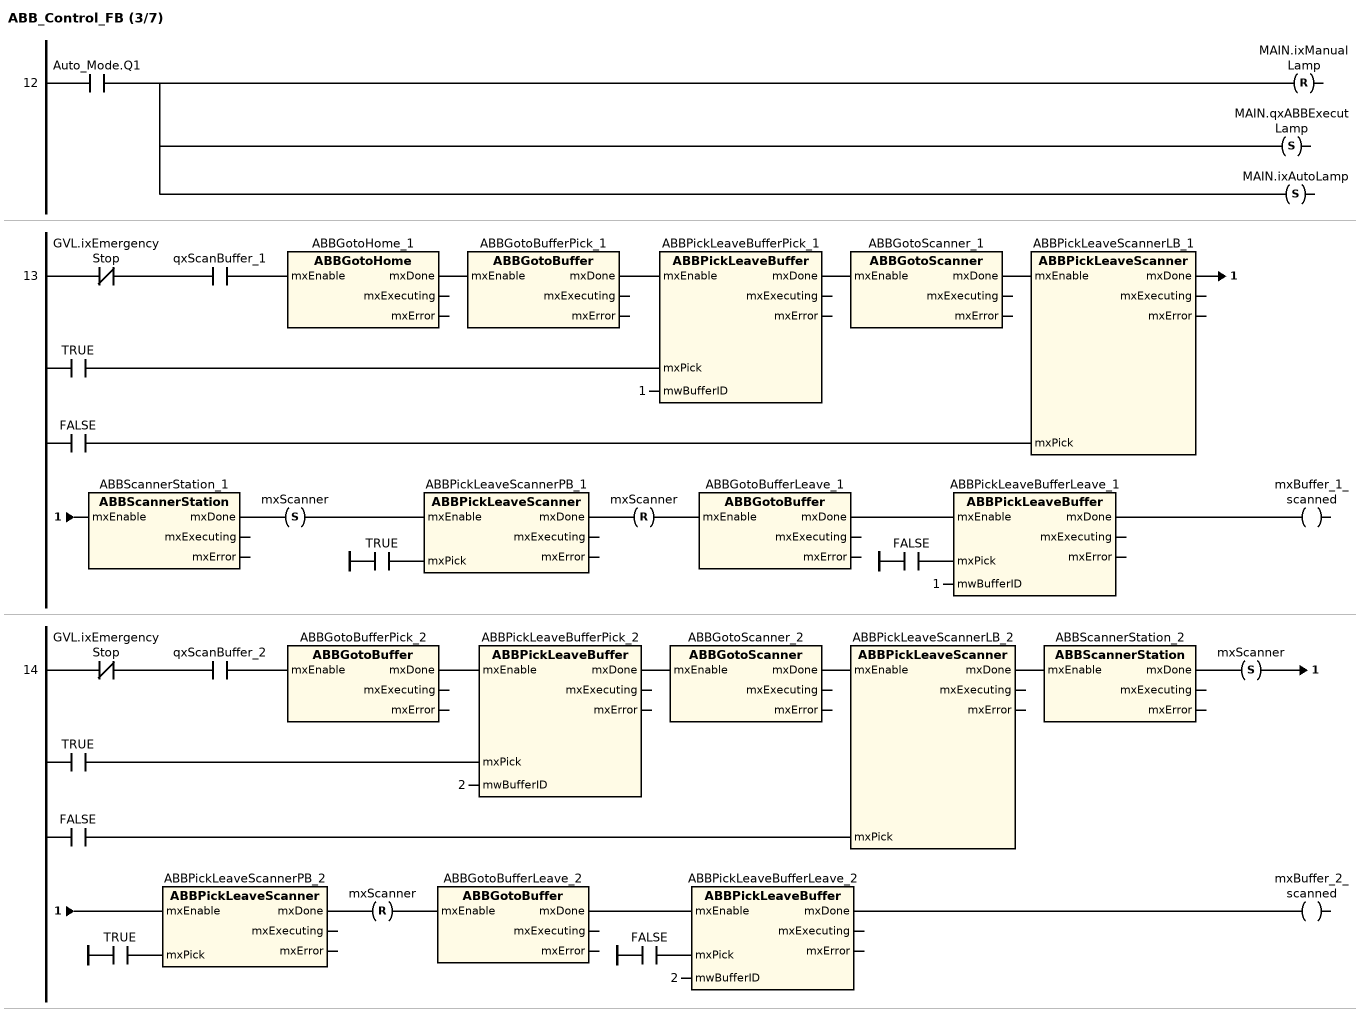
// NETWORK 12
MAIN.ixManualLamp R= Auto_Mode.Q1;
MAIN.qxABBExecutLamp S= Auto_Mode.Q1;
MAIN.ixAutoLamp S= Auto_Mode.Q1;

// NETWORK 13
ABBGotoHome_1(mxEnable := NOT GVL.ixEmergencyStop AND qxScanBuffer_1); // ABBGotoHome
ABBGotoBufferPick_1(mxEnable := ABBGotoHome_1.mxDone); // ABBGotoBuffer
ABBPickLeaveBufferPick_1(mxEnable := ABBGotoBufferPick_1.mxDone, mxPick := TRUE, mwBufferID := 1); // ABBPickLeaveBuffer
ABBGotoScanner_1(mxEnable := ABBPickLeaveBufferPick_1.mxDone); // ABBGotoScanner
ABBPickLeaveScannerLB_1(mxEnable := ABBGotoScanner_1.mxDone, mxPick := FALSE); // ABBPickLeaveScanner
ABBScannerStation_1(mxEnable := ABBPickLeaveScannerLB_1.mxDone); // ABBScannerStation
mxScanner S= ABBScannerStation_1.mxDone;
ABBPickLeaveScannerPB_1(mxEnable := ABBScannerStation_1.mxDone, mxPick := TRUE); // ABBPickLeaveScanner
mxScanner R= ABBPickLeaveScannerPB_1.mxDone;
ABBGotoBufferLeave_1(mxEnable := ABBPickLeaveScannerPB_1.mxDone); // ABBGotoBuffer
ABBPickLeaveBufferLeave_1(mxEnable := ABBGotoBufferLeave_1.mxDone, mxPick := FALSE, mwBufferID := 1); // ABBPickLeaveBuffer
mxBuffer_1_scanned := ABBPickLeaveBufferLeave_1.mxDone;

// NETWORK 14
ABBGotoBufferPick_2(mxEnable := NOT GVL.ixEmergencyStop AND qxScanBuffer_2); // ABBGotoBuffer
ABBPickLeaveBufferPick_2(mxEnable := ABBGotoBufferPick_2.mxDone, mxPick := TRUE, mwBufferID := 2); // ABBPickLeaveBuffer
ABBGotoScanner_2(mxEnable := ABBPickLeaveBufferPick_2.mxDone); // ABBGotoScanner
ABBPickLeaveScannerLB_2(mxEnable := ABBGotoScanner_2.mxDone, mxPick := FALSE); // ABBPickLeaveScanner
ABBScannerStation_2(mxEnable := ABBPickLeaveScannerLB_2.mxDone); // ABBScannerStation
mxScanner S= ABBScannerStation_2.mxDone;
ABBPickLeaveScannerPB_2(mxEnable := ABBScannerStation_2.mxDone, mxPick := TRUE); // ABBPickLeaveScanner
mxScanner R= ABBPickLeaveScannerPB_2.mxDone;
ABBGotoBufferLeave_2(mxEnable := ABBPickLeaveScannerPB_2.mxDone); // ABBGotoBuffer
ABBPickLeaveBufferLeave_2(mxEnable := ABBGotoBufferLeave_2.mxDone, mxPick := FALSE, mwBufferID := 2); // ABBPickLeaveBuffer
mxBuffer_2_scanned := ABBPickLeaveBufferLeave_2.mxDone;

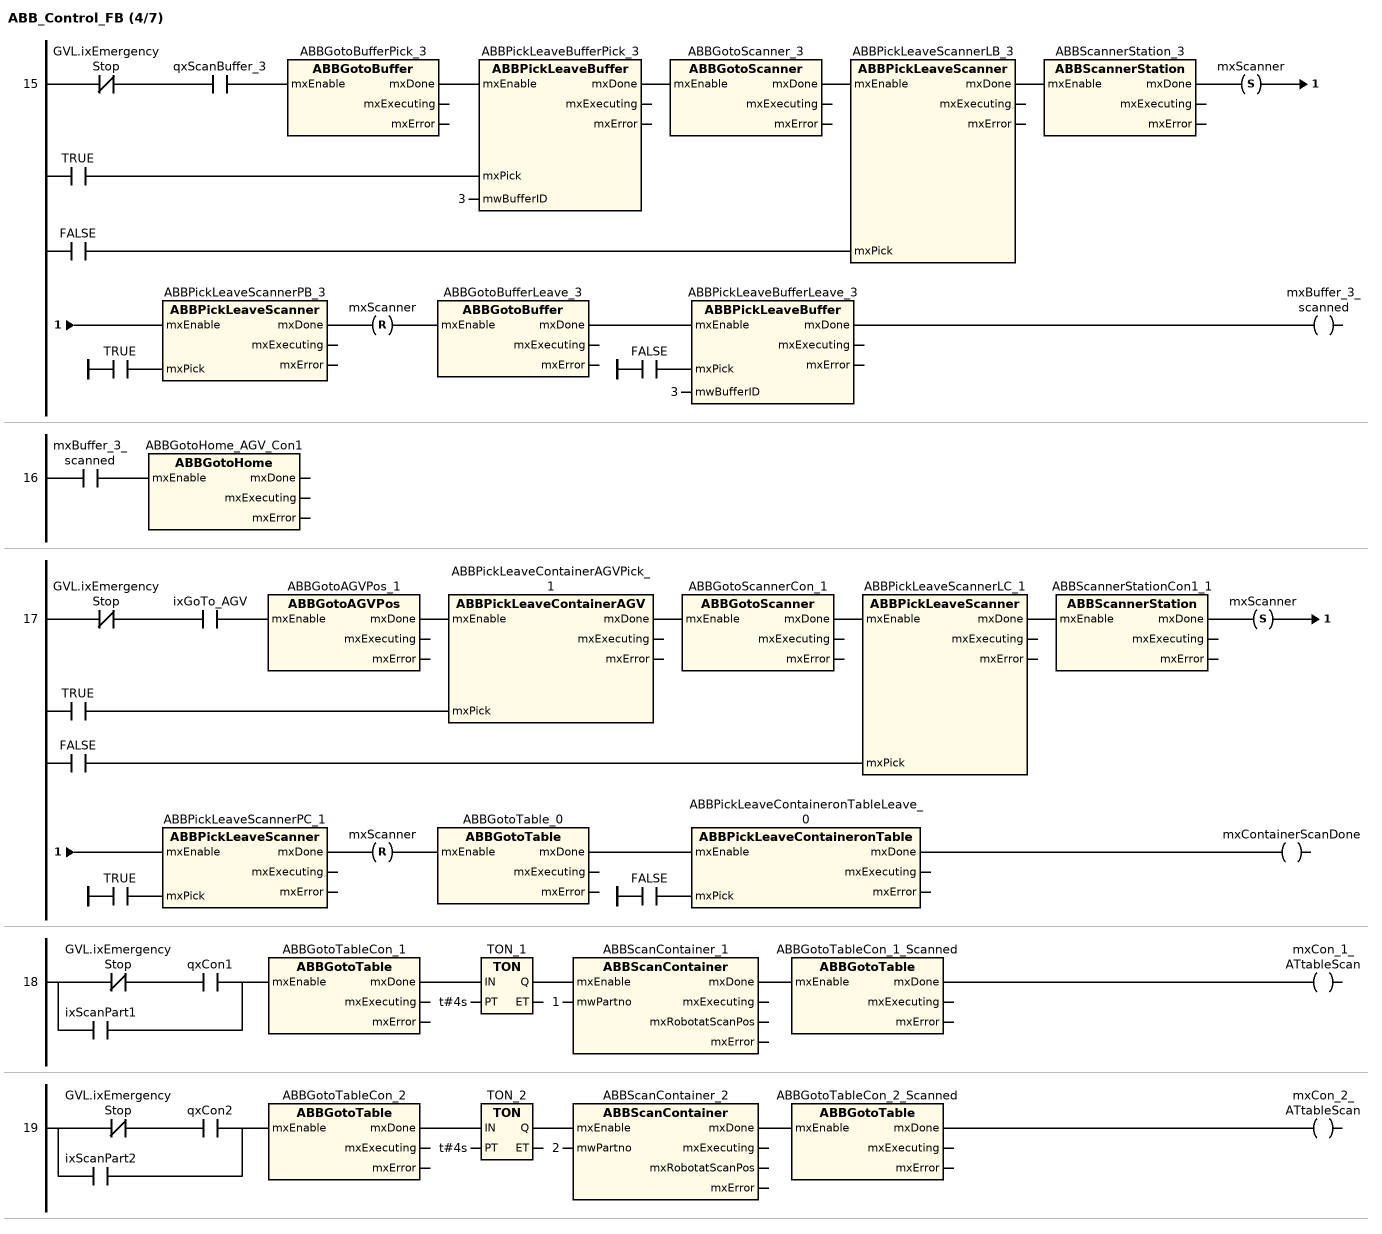
// NETWORK 15
ABBGotoBufferPick_3(mxEnable := NOT GVL.ixEmergencyStop AND qxScanBuffer_3); // ABBGotoBuffer
ABBPickLeaveBufferPick_3(mxEnable := ABBGotoBufferPick_3.mxDone, mxPick := TRUE, mwBufferID := 3); // ABBPickLeaveBuffer
ABBGotoScanner_3(mxEnable := ABBPickLeaveBufferPick_3.mxDone); // ABBGotoScanner
ABBPickLeaveScannerLB_3(mxEnable := ABBGotoScanner_3.mxDone, mxPick := FALSE); // ABBPickLeaveScanner
ABBScannerStation_3(mxEnable := ABBPickLeaveScannerLB_3.mxDone); // ABBScannerStation
mxScanner S= ABBScannerStation_3.mxDone;
ABBPickLeaveScannerPB_3(mxEnable := ABBScannerStation_3.mxDone, mxPick := TRUE); // ABBPickLeaveScanner
mxScanner R= ABBPickLeaveScannerPB_3.mxDone;
ABBGotoBufferLeave_3(mxEnable := ABBPickLeaveScannerPB_3.mxDone); // ABBGotoBuffer
ABBPickLeaveBufferLeave_3(mxEnable := ABBGotoBufferLeave_3.mxDone, mxPick := FALSE, mwBufferID := 3); // ABBPickLeaveBuffer
mxBuffer_3_scanned := ABBPickLeaveBufferLeave_3.mxDone;

// NETWORK 16
ABBGotoHome_AGV_Con1(mxEnable := mxBuffer_3_scanned); // ABBGotoHome

// NETWORK 17
ABBGotoAGVPos_1(mxEnable := NOT GVL.ixEmergencyStop AND ixGoTo_AGV); // ABBGotoAGVPos
ABBPickLeaveContainerAGVPick_1(mxEnable := ABBGotoAGVPos_1.mxDone, mxPick := TRUE); // ABBPickLeaveContainerAGV
ABBGotoScannerCon_1(mxEnable := ABBPickLeaveContainerAGVPick_1.mxDone); // ABBGotoScanner
ABBPickLeaveScannerLC_1(mxEnable := ABBGotoScannerCon_1.mxDone, mxPick := FALSE); // ABBPickLeaveScanner
ABBScannerStationCon1_1(mxEnable := ABBPickLeaveScannerLC_1.mxDone); // ABBScannerStation
mxScanner S= ABBScannerStationCon1_1.mxDone;
ABBPickLeaveScannerPC_1(mxEnable := ABBScannerStationCon1_1.mxDone, mxPick := TRUE); // ABBPickLeaveScanner
mxScanner R= ABBPickLeaveScannerPC_1.mxDone;
ABBGotoTable_0(mxEnable := ABBPickLeaveScannerPC_1.mxDone); // ABBGotoTable
ABBPickLeaveContaineronTableLeave_0(mxEnable := ABBGotoTable_0.mxDone, mxPick := FALSE); // ABBPickLeaveContaineronTable
mxContainerScanDone := ABBPickLeaveContaineronTableLeave_0.mxDone;

// NETWORK 18
ABBGotoTableCon_1(mxEnable := NOT GVL.ixEmergencyStop AND qxCon1 OR ixScanPart1); // ABBGotoTable
TON_1(IN := ABBGotoTableCon_1.mxDone, PT := t#4s); // TON
ABBScanContainer_1(mxEnable := TON_1.Q, mwPartno := 1); // ABBScanContainer
ABBGotoTableCon_1_Scanned(mxEnable := ABBScanContainer_1.mxDone); // ABBGotoTable
mxCon_1_ATtableScan := ABBGotoTableCon_1_Scanned.mxDone;

// NETWORK 19
ABBGotoTableCon_2(mxEnable := NOT GVL.ixEmergencyStop AND qxCon2 OR ixScanPart2); // ABBGotoTable
TON_2(IN := ABBGotoTableCon_2.mxDone, PT := t#4s); // TON
ABBScanContainer_2(mxEnable := TON_2.Q, mwPartno := 2); // ABBScanContainer
ABBGotoTableCon_2_Scanned(mxEnable := ABBScanContainer_2.mxDone); // ABBGotoTable
mxCon_2_ATtableScan := ABBGotoTableCon_2_Scanned.mxDone;

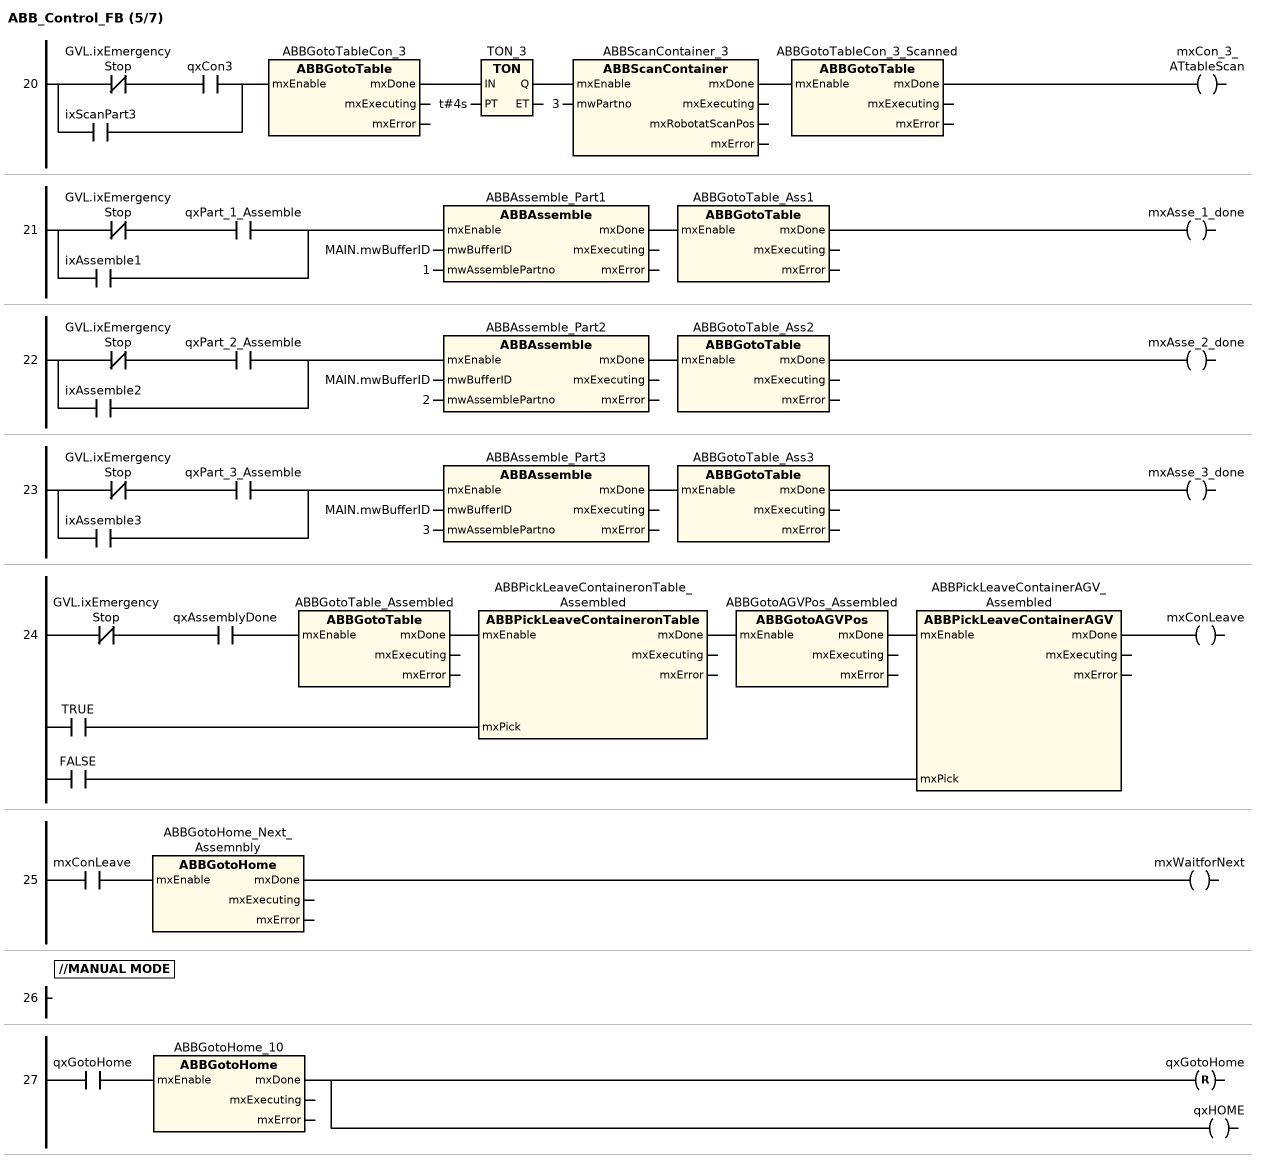
// NETWORK 20
ABBGotoTableCon_3(mxEnable := NOT GVL.ixEmergencyStop AND qxCon3 OR ixScanPart3); // ABBGotoTable
TON_3(IN := ABBGotoTableCon_3.mxDone, PT := t#4s); // TON
ABBScanContainer_3(mxEnable := TON_3.Q, mwPartno := 3); // ABBScanContainer
ABBGotoTableCon_3_Scanned(mxEnable := ABBScanContainer_3.mxDone); // ABBGotoTable
mxCon_3_ATtableScan := ABBGotoTableCon_3_Scanned.mxDone;

// NETWORK 21
ABBAssemble_Part1(
    mxEnable := NOT GVL.ixEmergencyStop AND qxPart_1_Assemble OR ixAssemble1,
    mwBufferID := MAIN.mwBufferID,
    mwAssemblePartno := 1); // ABBAssemble
ABBGotoTable_Ass1(mxEnable := ABBAssemble_Part1.mxDone); // ABBGotoTable
mxAsse_1_done := ABBGotoTable_Ass1.mxDone;

// NETWORK 22
ABBAssemble_Part2(
    mxEnable := NOT GVL.ixEmergencyStop AND qxPart_2_Assemble OR ixAssemble2,
    mwBufferID := MAIN.mwBufferID,
    mwAssemblePartno := 2); // ABBAssemble
ABBGotoTable_Ass2(mxEnable := ABBAssemble_Part2.mxDone); // ABBGotoTable
mxAsse_2_done := ABBGotoTable_Ass2.mxDone;

// NETWORK 23
ABBAssemble_Part3(
    mxEnable := NOT GVL.ixEmergencyStop AND qxPart_3_Assemble OR ixAssemble3,
    mwBufferID := MAIN.mwBufferID,
    mwAssemblePartno := 3); // ABBAssemble
ABBGotoTable_Ass3(mxEnable := ABBAssemble_Part3.mxDone); // ABBGotoTable
mxAsse_3_done := ABBGotoTable_Ass3.mxDone;

// NETWORK 24
ABBGotoTable_Assembled(mxEnable := NOT GVL.ixEmergencyStop AND qxAssemblyDone); // ABBGotoTable
ABBPickLeaveContaineronTable_Assembled(mxEnable := ABBGotoTable_Assembled.mxDone, mxPick := TRUE); // ABBPickLeaveContaineronTable
ABBGotoAGVPos_Assembled(mxEnable := ABBPickLeaveContaineronTable_Assembled.mxDone); // ABBGotoAGVPos
ABBPickLeaveContainerAGV_Assembled(mxEnable := ABBGotoAGVPos_Assembled.mxDone, mxPick := FALSE); // ABBPickLeaveContainerAGV
mxConLeave := ABBPickLeaveContainerAGV_Assembled.mxDone;

// NETWORK 25
ABBGotoHome_Next_Assemnbly(mxEnable := mxConLeave); // ABBGotoHome
mxWaitforNext := ABBGotoHome_Next_Assemnbly.mxDone;

// NETWORK 26
// label: //MANUAL MODE

// NETWORK 27
ABBGotoHome_10(mxEnable := qxGotoHome); // ABBGotoHome
qxGotoHome R= ABBGotoHome_10.mxDone;
qxHOME := ABBGotoHome_10.mxDone;

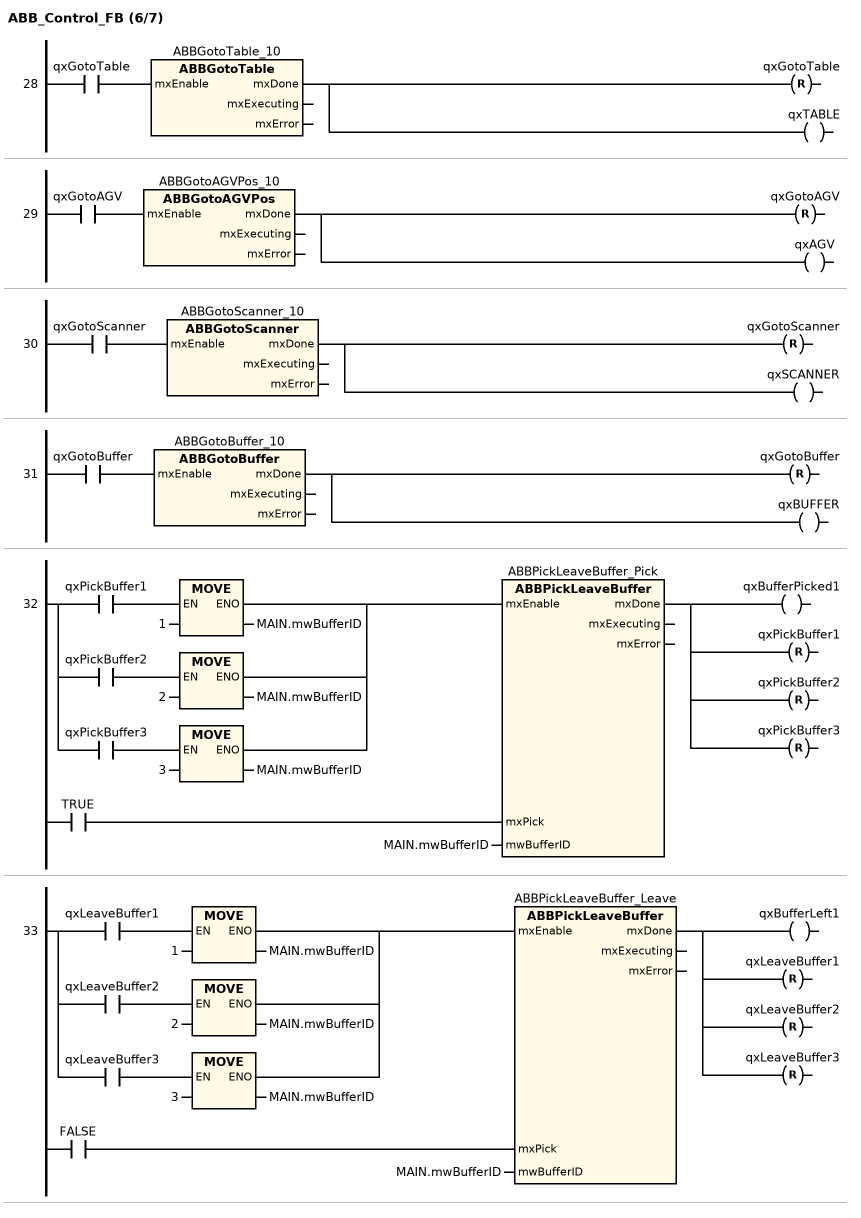
// NETWORK 28
ABBGotoTable_10(mxEnable := qxGotoTable); // ABBGotoTable
qxGotoTable R= ABBGotoTable_10.mxDone;
qxTABLE := ABBGotoTable_10.mxDone;

// NETWORK 29
ABBGotoAGVPos_10(mxEnable := qxGotoAGV); // ABBGotoAGVPos
qxGotoAGV R= ABBGotoAGVPos_10.mxDone;
qxAGV := ABBGotoAGVPos_10.mxDone;

// NETWORK 30
ABBGotoScanner_10(mxEnable := qxGotoScanner); // ABBGotoScanner
qxGotoScanner R= ABBGotoScanner_10.mxDone;
qxSCANNER := ABBGotoScanner_10.mxDone;

// NETWORK 31
ABBGotoBuffer_10(mxEnable := qxGotoBuffer); // ABBGotoBuffer
qxGotoBuffer R= ABBGotoBuffer_10.mxDone;
qxBUFFER := ABBGotoBuffer_10.mxDone;

// NETWORK 32
_w2 := qxPickBuffer1;
IF _w2 THEN MAIN.mwBufferID := 1; END_IF
_w3 := qxPickBuffer2;
IF _w3 THEN MAIN.mwBufferID := 2; END_IF
_w4 := qxPickBuffer3;
IF _w4 THEN MAIN.mwBufferID := 3; END_IF
ABBPickLeaveBuffer_Pick(mxEnable := _w2 OR _w3 OR _w4, mxPick := TRUE, mwBufferID := MAIN.mwBufferID); // ABBPickLeaveBuffer
qxBufferPicked1 := ABBPickLeaveBuffer_Pick.mxDone;
qxPickBuffer1 R= ABBPickLeaveBuffer_Pick.mxDone;
qxPickBuffer2 R= ABBPickLeaveBuffer_Pick.mxDone;
qxPickBuffer3 R= ABBPickLeaveBuffer_Pick.mxDone;

// NETWORK 33
_w5 := qxLeaveBuffer1;
IF _w5 THEN MAIN.mwBufferID := 1; END_IF
_w6 := qxLeaveBuffer2;
IF _w6 THEN MAIN.mwBufferID := 2; END_IF
_w7 := qxLeaveBuffer3;
IF _w7 THEN MAIN.mwBufferID := 3; END_IF
ABBPickLeaveBuffer_Leave(mxEnable := _w5 OR _w6 OR _w7, mxPick := FALSE, mwBufferID := MAIN.mwBufferID); // ABBPickLeaveBuffer
qxBufferLeft1 := ABBPickLeaveBuffer_Leave.mxDone;
qxLeaveBuffer1 R= ABBPickLeaveBuffer_Leave.mxDone;
qxLeaveBuffer2 R= ABBPickLeaveBuffer_Leave.mxDone;
qxLeaveBuffer3 R= ABBPickLeaveBuffer_Leave.mxDone;

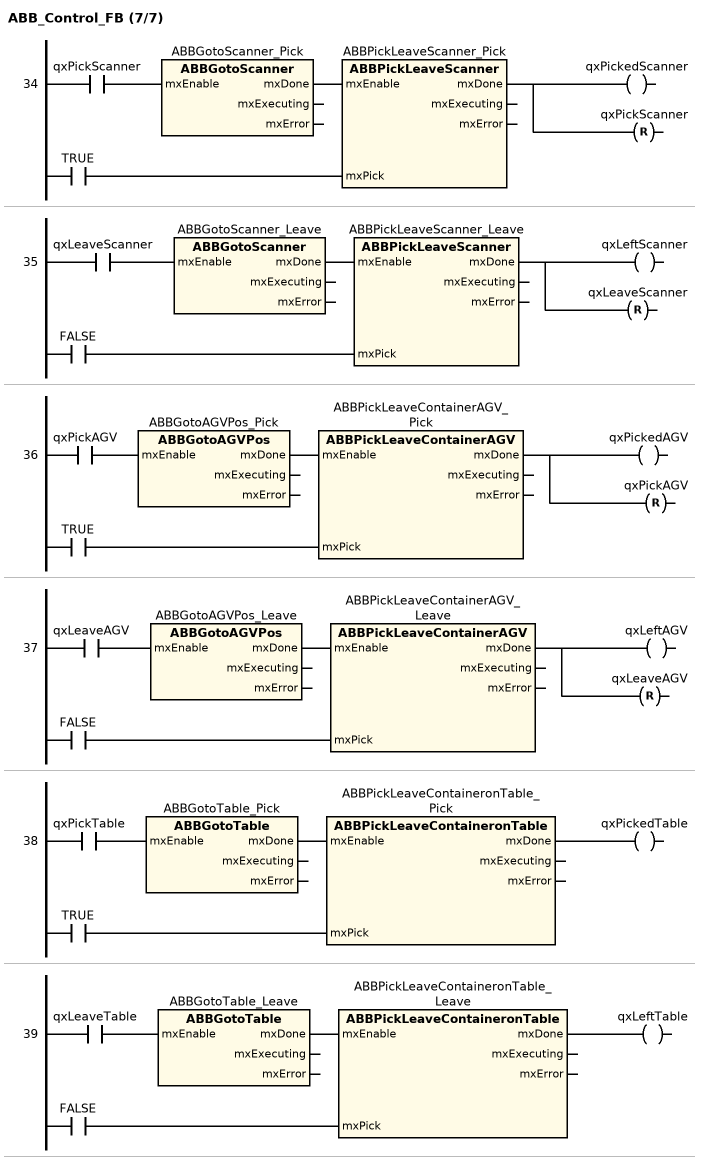
// NETWORK 34
ABBGotoScanner_Pick(mxEnable := qxPickScanner); // ABBGotoScanner
ABBPickLeaveScanner_Pick(mxEnable := ABBGotoScanner_Pick.mxDone, mxPick := TRUE); // ABBPickLeaveScanner
qxPickedScanner := ABBPickLeaveScanner_Pick.mxDone;
qxPickScanner R= ABBPickLeaveScanner_Pick.mxDone;

// NETWORK 35
ABBGotoScanner_Leave(mxEnable := qxLeaveScanner); // ABBGotoScanner
ABBPickLeaveScanner_Leave(mxEnable := ABBGotoScanner_Leave.mxDone, mxPick := FALSE); // ABBPickLeaveScanner
qxLeftScanner := ABBPickLeaveScanner_Leave.mxDone;
qxLeaveScanner R= ABBPickLeaveScanner_Leave.mxDone;

// NETWORK 36
ABBGotoAGVPos_Pick(mxEnable := qxPickAGV); // ABBGotoAGVPos
ABBPickLeaveContainerAGV_Pick(mxEnable := ABBGotoAGVPos_Pick.mxDone, mxPick := TRUE); // ABBPickLeaveContainerAGV
qxPickedAGV := ABBPickLeaveContainerAGV_Pick.mxDone;
qxPickAGV R= ABBPickLeaveContainerAGV_Pick.mxDone;

// NETWORK 37
ABBGotoAGVPos_Leave(mxEnable := qxLeaveAGV); // ABBGotoAGVPos
ABBPickLeaveContainerAGV_Leave(mxEnable := ABBGotoAGVPos_Leave.mxDone, mxPick := FALSE); // ABBPickLeaveContainerAGV
qxLeftAGV := ABBPickLeaveContainerAGV_Leave.mxDone;
qxLeaveAGV R= ABBPickLeaveContainerAGV_Leave.mxDone;

// NETWORK 38
ABBGotoTable_Pick(mxEnable := qxPickTable); // ABBGotoTable
ABBPickLeaveContaineronTable_Pick(mxEnable := ABBGotoTable_Pick.mxDone, mxPick := TRUE); // ABBPickLeaveContaineronTable
qxPickedTable := ABBPickLeaveContaineronTable_Pick.mxDone;

// NETWORK 39
ABBGotoTable_Leave(mxEnable := qxLeaveTable); // ABBGotoTable
ABBPickLeaveContaineronTable_Leave(mxEnable := ABBGotoTable_Leave.mxDone, mxPick := FALSE); // ABBPickLeaveContaineronTable
qxLeftTable := ABBPickLeaveContaineronTable_Leave.mxDone;

END_PROGRAM

// ---- ABBControl/ABBGotoBuffer.TcPOU
FUNCTION_BLOCK ABBGotoBuffer
VAR_INPUT
	mxEnable: BOOL;
END_VAR
VAR_OUTPUT
	mxDone:BOOL;
	mxExecuting: BOOL;
	mxError: BOOL;
END_VAR
VAR
	ABB: INT;
END_VAR

CASE ABB OF
	0:
		IF mxEnable AND NOT CommData.mxABBExecuting THEN
			ABB:=10;
		END_IF
	10:
		IF CommData.mxRobotOnline THEN
			ABB:=100;
			ELSE
			ABB:=200;
		END_IF
	100:
		mxExecuting:=TRUE;
		CommData.maOrderMaker[1] := 1;
		CommData.maOrderMaker[2] := 0;
		CommData.maOrderMaker[3] := 0;
		CommData.maOrderMaker[4] := 0;
		CommData.maOrderMaker[5] := 0;
		CommData.maOrderMaker[6] := 5;
		CommData.qwOrderRobot:=100005;
		ABB:=101;
	101:
		IF CommData.qwOrderRobot > 0 THEN
			CommData.qxPLCStrobe:=TRUE;
			ABB:=102;
		END_IF
	102:
		IF CommData.ixRobotStrobe THEN
			IF CommData.iwReplyRobot = CommData.qwOrderRobot+1 THEN
				CommData.qwOrderRobot:=0;
				CommData.maOrderMaker[1] := 0;
				CommData.maOrderMaker[2] := 0;
				CommData.maOrderMaker[3] := 0;
				CommData.maOrderMaker[4] := 0;
				CommData.maOrderMaker[5] := 0;
				CommData.maOrderMaker[6] := 0;
				CommData.qxPLCStrobe:=FALSE;
				ABB:=103;
			ELSE
				ABB:=1000;
			END_IF
		END_IF
	103:
		IF NOT CommData.ixRobotStrobe THEN
			IF CommData.iwReplyRobot = 0 THEN
				ABB:=104;
			ELSE
				ABB:=1000;
			END_IF
		END_IF
	104:
		IF CommData.ixRobotStrobe THEN
			IF CommData.iwProgressRobot = 90 THEN
				CommData.qxPLCStrobe:=TRUE;
				ABB:=105;
			END_IF
			IF CommData.iwProgressRobot = 1000 THEN
				CommData.qxPLCStrobe:=TRUE;
				ABB:=1000;
			END_IF
		END_IF	
	105:
		IF  NOT CommData.ixRobotStrobe AND CommData.iwProgressRobot = 0 THEN
			CommData.qxPLCStrobe:=FALSE;
			ABB:=201;
		END_IF	
		
	200:
		CommData.mwABBPosXaxis:=CommData.ABBPostions.Bufferhome.X;
		CommData.mwABBPosYaxis:=CommData.ABBPostions.Bufferhome.Y;
		mxExecuting:=TRUE;
		CommData.mxStartABB:=TRUE;
		IF CommData.mwXaxis = CommData.ABBPostions.Bufferhome.X AND CommData.mwYaxis = CommData.ABBPostions.Bufferhome.Y THEN
			ABB:=201;
		ELSIF gvl.ixEmergencyStop THEN
			ABB:=1000;
		END_IF
	201:
		mxExecuting:=FALSE;
		CommData.mxStartABB:=FALSE;
		mxDone:=TRUE;
		IF NOT mxEnable THEN
			mxDone:=FALSE;
			ABB:=0;
		END_IF
	1000:
		mxError:=TRUE;
		mxExecuting:=FALSE;
		CommData.mxStartABB:=FALSE;
		IF NOT mxEnable THEN
			mxError:=FALSE;
			mxDone:=FALSE;
			ABB:=0;
		END_IF
END_CASE




IF gvl.ixEmergencyStop THEN
	ABB:=1000;
END_IF

END_FUNCTION_BLOCK

// ---- ABBControl/ABBPickLeaveBuffer.TcPOU
FUNCTION_BLOCK ABBPickLeaveBuffer
VAR_INPUT
	mxEnable: BOOL;
	mxPick: BOOL;
	mwBufferID: INT;
END_VAR
VAR_OUTPUT
	mxDone: BOOL;
	mxExecuting: BOOL;
	mxError: BOOL;
END_VAR
VAR
	ABB: INT;
	mwordernumber: DINT;
END_VAR

CASE ABB OF
		0:
			IF mxEnable AND NOT CommData.mxABBExecuting THEN
				ABB:=1;
			END_IF
		1:
			IF CommData.mxRobotOnline THEN
				ABB:=100;
				ELSE
				ABB:=200;
			END_IF
		100:
			IF CommData.msRobotLastPos = 'Buffer' THEN
				ABB:=101;
			ELSE
				ABB:=1000;
			END_IF
		101:
			mxExecuting:=TRUE;
			CommData.maOrderMaker[1] := 9;
			CommData.maOrderMaker[4] := 0;
			CommData.maOrderMaker[5] := 0;
			CommData.maOrderMaker[6] := 0;
			ABB:=102;
		102:
			IF mxPick THEN
				CommData.maOrderMaker[2] := 1;
				ABB:=1021;
			ELSIF NOT mxPick THEN
				CommData.maOrderMaker[2] := 0;
				ABB:=1021;
			END_IF
		1021:
			IF mwBufferID = 1 OR mwBufferID = 2 OR mwBufferID = 3 THEN
				CommData.maOrderMaker[3] := mwBufferID;
				ABB:=103;
			ELSE
				ABB:=1000;//Error
			END_IF
		103:
				mwordernumber:=CommData.maOrderMaker[1];
				mwordernumber:=mwordernumber*10;
				abb:=1151;
		1151:
				mwordernumber:=mwordernumber+CommData.maOrderMaker[2];
				abb:=1152;
		1152:
				mwordernumber:=mwordernumber*10;
				abb:=1153;
		1153:
				mwordernumber:=mwordernumber+CommData.maOrderMaker[3];
				abb:=1154;
		1154:
				mwordernumber:=mwordernumber*10;
				abb:=1155;
		1155:
				mwordernumber:=mwordernumber+CommData.maOrderMaker[4];
				abb:=1156;
		1156:
				mwordernumber:=mwordernumber*10;
				abb:=1157;
		1157:
				mwordernumber:=mwordernumber+CommData.maOrderMaker[5];
				abb:=1158;
		1158:
				mwordernumber:=mwordernumber*10;
				abb:=1159;
		1159:
				mwordernumber:=mwordernumber+CommData.maOrderMaker[6];
				ABB:=1160;
		1160:
			CommData.qwOrderRobot:=mwordernumber;
			ABB:=104;
		104:
			IF CommData.qwOrderRobot > 0 THEN
				CommData.qxPLCStrobe:=TRUE;
				ABB:=105;
			END_IF
		105:
			IF CommData.ixRobotStrobe THEN
				IF CommData.iwReplyRobot = CommData.qwOrderRobot+1 THEN
					CommData.qwOrderRobot:=0;
					mwordernumber:=0;
					CommData.qxPLCStrobe:=FALSE;
					ABB:=106;
				ELSE
					ABB:=1000;
				END_IF
			END_IF
		106:
			IF NOT CommData.ixRobotStrobe THEN
				IF CommData.iwReplyRobot = 0 THEN
						ABB:=107;
					ELSE
						ABB:=1000;
				END_IF
			END_IF
		107:
			IF CommData.ixRobotStrobe THEN
				IF CommData.iwProgressRobot = 90 THEN
					CommData.qxPLCStrobe:=TRUE;
					ABB:=108;
				END_IF
				IF CommData.iwProgressRobot = 1000 THEN
					CommData.qxPLCStrobe:=TRUE;
					ABB:=1000;
				END_IF
			END_IF
		108:
			IF  NOT CommData.ixRobotStrobe AND CommData.iwProgressRobot = 0 THEN
				CommData.qxPLCStrobe:=FALSE;
				ABB:=33;
			END_IF
	
		
		
		200:
			IF mwBufferID = 1 THEN
				ABB:=10;
			ELSIF mwBufferID = 2 THEN
				ABB:=20;
			ELSIF mwBufferID = 3 THEN
				ABB:=30;
			ELSE
				ABB:=1000;//Error
			END_IF
		10:
			IF CommData.mwXaxis = CommData.ABBPostions.Bufferhome.X AND CommData.mwYaxis = CommData.ABBPostions.Bufferhome.Y THEN
				ABB:=11;
			ELSE
				ABB:=1000;
			END_IF
		11:
			CommData.mwABBPosXaxis:=CommData.ABBPostions.Storage1.X;
			CommData.mwABBPosYaxis:=CommData.ABBPostions.Storage1.Y;
			mxExecuting:=TRUE;
			CommData.mxStartABB:=TRUE;
			IF CommData.mwXaxis = CommData.ABBPostions.Storage1.X AND CommData.mwYaxis = CommData.ABBPostions.Storage1.Y THEN
				CommData.mxStartABB:=FALSE;
				ABB:=12;
			ELSIF gvl.ixEmergencyStop THEN
				ABB:=1000;
			END_IF
		12:
			IF mxpick THEN
				IF NOT CommData.mxGripper THEN
					CommData.mxGripper:=TRUE;
					ABB:=13;
				ELSE
					ABB:=1000;
				END_IF
			ELSIF NOT mxPick THEN
				IF CommData.mxGripper THEN
					CommData.mxGripper:=FALSE;
					ABB:=13;
				ELSE
					ABB:=1000;
				END_IF
			END_IF
		13:
			mxExecuting:=FALSE;
			mxDone:=TRUE;
			IF NOT mxEnable THEN
				mxError:=FALSE;
				mxDone:=FALSE;
				ABB:=0;
			END_IF
		
		20:
			IF CommData.mwXaxis = CommData.ABBPostions.Bufferhome.X AND CommData.mwYaxis = CommData.ABBPostions.Bufferhome.Y THEN
				ABB:=21;
			ELSE
				ABB:=1000;
			END_IF
		21:
			CommData.mwABBPosXaxis:=CommData.ABBPostions.Storage2.X;
			CommData.mwABBPosYaxis:=CommData.ABBPostions.Storage2.Y;
			mxExecuting:=TRUE;
			CommData.mxStartABB:=TRUE;
			IF CommData.mwXaxis = CommData.ABBPostions.Storage2.X AND CommData.mwYaxis = CommData.ABBPostions.Storage2.Y THEN
				CommData.mxStartABB:=FALSE;
				ABB:=22;
			ELSIF gvl.ixEmergencyStop THEN
				ABB:=1000;
			END_IF
		22:
			IF mxpick THEN
				IF NOT CommData.mxGripper THEN
					CommData.mxGripper:=TRUE;
					ABB:=23;
				ELSE
					ABB:=1000;
				END_IF
			ELSIF NOT mxPick THEN
				IF CommData.mxGripper THEN
					CommData.mxGripper:=FALSE;
					ABB:=23;
				ELSE
					ABB:=1000;
				END_IF
			END_IF
		23:
			mxExecuting:=FALSE;
			mxDone:=TRUE;
			IF NOT mxEnable THEN
				mxError:=FALSE;
				mxDone:=FALSE;
				ABB:=0;
			END_IF
		

		30:
			IF CommData.mwXaxis = CommData.ABBPostions.Bufferhome.X AND CommData.mwYaxis = CommData.ABBPostions.Bufferhome.Y THEN
				ABB:=31;
			ELSE
				ABB:=1000;
			END_IF
		31:
			CommData.mwABBPosXaxis:=CommData.ABBPostions.Storage3.X;
			CommData.mwABBPosYaxis:=CommData.ABBPostions.Storage3.Y;
			mxExecuting:=TRUE;
			CommData.mxStartABB:=TRUE;
			IF CommData.mwXaxis = CommData.ABBPostions.Storage3.X AND CommData.mwYaxis = CommData.ABBPostions.Storage3.Y THEN
				CommData.mxStartABB:=FALSE;
				ABB:=32;
			ELSIF gvl.ixEmergencyStop THEN
				ABB:=1000;
			END_IF
		32:
			IF mxpick THEN
				IF NOT CommData.mxGripper THEN
					CommData.mxGripper:=TRUE;
					ABB:=33;
				ELSE
					ABB:=1000;
				END_IF
			ELSIF NOT mxPick THEN
				IF CommData.mxGripper THEN
					CommData.mxGripper:=FALSE;
					ABB:=33;
				ELSE
					ABB:=1000;
				END_IF
			END_IF
		33:
			mxExecuting:=FALSE;
			mxDone:=TRUE;
			IF NOT mxEnable THEN
				mxError:=FALSE;
				mxDone:=FALSE;
				ABB:=0;
			END_IF	

		1000:
			mxError:=TRUE;
			IF NOT mxEnable THEN
				mxError:=FALSE;
				mxDone:=FALSE;
				ABB:=0;
			END_IF
END_CASE



IF gvl.ixEmergencyStop THEN
	ABB:=1000;
END_IF

END_FUNCTION_BLOCK

// ---- ABBControl/ABBGotoScanner.TcPOU
FUNCTION_BLOCK ABBGotoScanner
VAR_INPUT
	mxEnable: BOOL;
END_VAR
VAR_OUTPUT
	mxDone:BOOL;
	mxExecuting: BOOL;
	mxError: BOOL;
END_VAR
VAR
	ABB: INT;
END_VAR

CASE ABB OF
	0:
		IF mxEnable AND NOT CommData.mxABBExecuting THEN
			ABB:=10;
		END_IF	
	10:
		IF CommData.mxRobotOnline THEN
			ABB:=100;
			ELSE
			ABB:=200;
		END_IF
	100:
		mxExecuting:=TRUE;
		CommData.maOrderMaker[1] := 2;
		CommData.maOrderMaker[2] := 0;
		CommData.maOrderMaker[3] := 0;
		CommData.maOrderMaker[4] := 0;
		CommData.maOrderMaker[5] := 0;
		CommData.maOrderMaker[6] := 5;
		CommData.qwOrderRobot:=200005;
		ABB:=101;
	101:
		IF CommData.qwOrderRobot > 0 THEN
			CommData.qxPLCStrobe:=TRUE;
			ABB:=102;
		END_IF
	102:
		IF CommData.ixRobotStrobe THEN
			IF CommData.iwReplyRobot = CommData.qwOrderRobot+1 THEN
				CommData.qwOrderRobot:=0;
				CommData.maOrderMaker[1] := 0;
				CommData.maOrderMaker[2] := 0;
				CommData.maOrderMaker[3] := 0;
				CommData.maOrderMaker[4] := 0;
				CommData.maOrderMaker[5] := 0;
				CommData.maOrderMaker[6] := 0;
				CommData.qxPLCStrobe:=FALSE;
				ABB:=103;
			ELSE
				ABB:=1000;
			END_IF
		END_IF
	103:
		IF NOT CommData.ixRobotStrobe THEN
			IF CommData.iwReplyRobot = 0 THEN
				ABB:=104;
			ELSE
				ABB:=1000;
			END_IF
		END_IF
	104:
		IF CommData.ixRobotStrobe THEN
			IF CommData.iwProgressRobot = 90 THEN
				CommData.qxPLCStrobe:=TRUE;
				ABB:=105;
			END_IF
			IF CommData.iwProgressRobot = 1000 THEN
				CommData.qxPLCStrobe:=TRUE;
				ABB:=1000;
			END_IF
		END_IF	
	105:
		IF  NOT CommData.ixRobotStrobe AND CommData.iwProgressRobot = 0 THEN
			CommData.qxPLCStrobe:=FALSE;
			ABB:=201;
		END_IF
		
		
	200:
		CommData.mwABBPosXaxis:=CommData.ABBPostions.Scannerhome.X;
		CommData.mwABBPosYaxis:=CommData.ABBPostions.Scannerhome.Y;
		mxExecuting:=TRUE;
		CommData.mxStartABB:=TRUE;
		IF CommData.mwXaxis = CommData.ABBPostions.Scannerhome.X AND CommData.mwYaxis = CommData.ABBPostions.Scannerhome.Y THEN
			ABB:=201;
		ELSIF gvl.ixEmergencyStop THEN
			ABB:=1000;
		END_IF
	201:
		mxExecuting:=FALSE;
		CommData.mxStartABB:=FALSE;
		mxDone:=TRUE;
		IF NOT mxEnable THEN
			mxDone:=FALSE;
			ABB:=0;
		END_IF
	1000:
		mxError:=TRUE;
		mxExecuting:=FALSE;
		CommData.mxStartABB:=FALSE;
		IF NOT mxEnable THEN
			mxError:=FALSE;
			mxDone:=FALSE;
			ABB:=0;
		END_IF
END_CASE



IF gvl.ixEmergencyStop THEN
	ABB:=1000;
END_IF

END_FUNCTION_BLOCK

// ---- ABBControl/ABBPickLeaveScanner.TcPOU
FUNCTION_BLOCK ABBPickLeaveScanner
VAR_INPUT
	mxEnable: BOOL;
	mxPick: BOOL;
END_VAR
VAR_OUTPUT
	mxDone:BOOL;
	mxExecuting: BOOL;
	mxError: BOOL;
END_VAR
VAR
	ABB: INT;
	mwordernumber: DINT;
END_VAR

CASE ABB OF
	0:
		IF mxEnable AND NOT CommData.mxABBExecuting THEN
			ABB:=10;
		END_IF
	10:
		IF CommData.mxRobotOnline THEN
			ABB:=100;
			ELSE
			ABB:=200;
		END_IF
	100:
		IF CommData.msRobotLastPos = 'Scanner' THEN
			ABB:=101;
		ELSE
			ABB:=1000;
		END_IF
	101:
		mxExecuting:=TRUE;
		CommData.maOrderMaker[1] := 6;
		CommData.maOrderMaker[3] := 0;
		CommData.maOrderMaker[4] := 0;
		CommData.maOrderMaker[5] := 0;
		CommData.maOrderMaker[6] := 0;
		ABB:=102;
	102:
		IF mxPick THEN
			CommData.maOrderMaker[2] := 1;
			ABB:=103;
		ELSIF NOT mxPick THEN
			CommData.maOrderMaker[2] := 0;
			ABB:=103;
		END_IF
	103:
		mwordernumber:=CommData.maOrderMaker[1];
			mwordernumber:=mwordernumber*10;
			abb:=1151;
	1151:
			mwordernumber:=mwordernumber+CommData.maOrderMaker[2];
			abb:=1152;
	1152:
			mwordernumber:=mwordernumber*10;
			abb:=1153;
	1153:
			mwordernumber:=mwordernumber+CommData.maOrderMaker[3];
			abb:=1154;
	1154:
			mwordernumber:=mwordernumber*10;
			abb:=1155;
	1155:
			mwordernumber:=mwordernumber+CommData.maOrderMaker[4];
			abb:=1156;
	1156:
			mwordernumber:=mwordernumber*10;
			abb:=1157;
	1157:
			mwordernumber:=mwordernumber+CommData.maOrderMaker[5];
			abb:=1158;
	1158:
			mwordernumber:=mwordernumber*10;
			abb:=1159;
	1159:
			mwordernumber:=mwordernumber+CommData.maOrderMaker[6];
			ABB:=1160;
	1160:
		CommData.qwOrderRobot:=mwordernumber;
		ABB:=104;
	104:
		IF CommData.qwOrderRobot > 0 THEN
			CommData.qxPLCStrobe:=TRUE;
			ABB:=105;
		END_IF
	105:
		IF CommData.ixRobotStrobe THEN
			IF CommData.iwReplyRobot = CommData.qwOrderRobot+1 THEN
				CommData.qwOrderRobot:=0;
				mwordernumber:=0;
				CommData.qxPLCStrobe:=FALSE;
				ABB:=106;
			ELSE
				ABB:=1000;
			END_IF
		END_IF
	106:
		IF NOT CommData.ixRobotStrobe THEN
			IF CommData.iwReplyRobot = 0 THEN
				ABB:=107;
			ELSE
				ABB:=1000;
			END_IF
		END_IF
	107:
		IF CommData.ixRobotStrobe THEN
			IF CommData.iwProgressRobot = 90 THEN
				CommData.qxPLCStrobe:=TRUE;
				ABB:=108;
			END_IF
			IF CommData.iwProgressRobot = 1000 THEN
				CommData.qxPLCStrobe:=TRUE;
				ABB:=1000;
			END_IF
		END_IF
	108:
		IF  NOT CommData.ixRobotStrobe AND CommData.iwProgressRobot = 0 THEN
			CommData.qxPLCStrobe:=FALSE;
			ABB:=202;
		END_IF
		
		
		
	200:
		mxExecuting:=TRUE;
		IF CommData.mwXaxis = CommData.ABBPostions.Scannerhome.X AND CommData.mwYaxis = CommData.ABBPostions.Scannerhome.Y THEN
			ABB:=201;
		ELSE
			ABB:=1000;
		END_IF
	201:
		IF mxpick THEN
			IF NOT CommData.mxGripper THEN
				CommData.mxGripper:=TRUE;
				ABB:=202;
			ELSE
				ABB:=1000;
			END_IF
		ELSIF NOT mxPick THEN
			IF CommData.mxGripper THEN
				CommData.mxGripper:=FALSE;
				ABB:=202;
			ELSE
				ABB:=1000;
			END_IF
		END_IF
	202:
		mxExecuting:=FALSE;
		mxDone:=TRUE;
		IF NOT mxEnable THEN
			mxError:=FALSE;
			mxDone:=FALSE;
			ABB:=0;
		END_IF
	1000:
		mxError:=TRUE;
		mxExecuting:=FALSE;
		IF NOT mxEnable THEN
			mxError:=FALSE;
			mxDone:=FALSE;
			ABB:=0;
		END_IF
END_CASE



IF gvl.ixEmergencyStop THEN
	ABB:=1000;
END_IF

END_FUNCTION_BLOCK

// ---- Automation Library/SensorReader.TcPOU
FUNCTION_BLOCK SensorReader
VAR_INPUT
	mxEnable: BOOL;
END_VAR
VAR_OUTPUT
	Product:STRING;
END_VAR
VAR
	SensorReader:BYTE;
END_VAR

IF mxEnable THEN
	SensorReader.1:=gvl.ixInductiveSensor1;
	SensorReader.2:=gvl.ixInductiveSensor2;
	SensorReader.3:=gvl.ixInductiveSensor3;
	SensorReader.4:=gvl.ixInductiveSensor4;
END_IF

IF SensorReader = 0 OR SensorReader = 4 OR SensorReader = 2 OR SensorReader = 6 THEN
 	Product:='InvalidPart';
END_IF

IF SensorReader=16 THEN
	Product:='Blue Container';
END_IF

IF SensorReader=8 THEN
	Product:='Yellow Container';
END_IF

IF SensorReader=24 THEN
	Product:='Red Container';
END_IF

IF SensorReader=20 THEN
	Product:='Blue Cylinder';
END_IF

IF SensorReader=12 THEN
	Product:='Blue Octagon';
END_IF

IF SensorReader=28 THEN
	Product:='Blue Plate';
END_IF

IF SensorReader=18 THEN
	Product:='Yellow Cylinder';
END_IF

IF SensorReader=10 THEN
	Product:='Yellow Octagon';
END_IF

IF SensorReader=26 THEN
	Product:='Yellow Plate';
END_IF

IF SensorReader=22 THEN
	Product:='Red Cylinder';
END_IF

IF SensorReader=14 THEN
	Product:='Red Octagon';
END_IF

IF SensorReader=30 THEN
	Product:='Red Plate';
END_IF

END_FUNCTION_BLOCK

// ---- ABBControl/ABBScannerStation.TcPOU
FUNCTION_BLOCK ABBScannerStation
VAR_INPUT
	mxEnable: BOOL;
END_VAR
VAR_OUTPUT
	mxDone:BOOL;
	mxExecuting: BOOL;
	mxError: BOOL;
END_VAR
VAR
	ABB: INT;
	mxWaitingforsensorinput: BOOL;
END_VAR

CASE ABB OF
	0:
		IF mxEnable THEN
			ABB:=10;
		END_IF
	10:
		IF (CommData.mwXaxis = CommData.ABBPostions.Scannerhome.X AND CommData.mwYaxis = CommData.ABBPostions.Scannerhome.Y) OR CommData.msRobotLastPos = 'Scanner'  THEN
			ABB:=20;
		ELSIF CommData.mxRobotOnline THEN
			ABB:=30;
		ELSE
			ABB:=1000;
		END_IF
	20:
		IF CommData.mxRobotOnline THEN
			ABB:=30;
		ELSE
			mxExecuting:=TRUE;
			commdata.mxWaitingforSensorinput:=TRUE;
			IF CommData.mxScannernoobject THEN
				ABB:=30;
			END_IF
		END_IF	
	30:
		commdata.mxWaitingforSensorinput:=FALSE;
		mxExecuting:=FALSE;
		mxDone:=TRUE;
		IF NOT mxEnable THEN
			mxDone:=FALSE;
			ABB:=0;
		END_IF
	1000:
		mxExecuting:=FALSE;
		mxError:=TRUE;
		IF NOT mxEnable THEN
			mxError:=FALSE;
			mxDone:=FALSE;
			ABB:=0;
		END_IF
		
END_CASE



IF gvl.ixEmergencyStop THEN
	ABB:=1000;
END_IF

END_FUNCTION_BLOCK

// ---- POUs/Scanner_FB.TcPOU
FUNCTION_BLOCK Scanner_FB
VAR_INPUT
	mxEnable: BOOL;
	mxRP: BOOL;
	mxYP: BOOL;
	mxBP: BOOL;
	mxRCy: BOOL;
	mxYCy: BOOL;
	mxBCy: BOOL;
	mxYOct: BOOL;
	mxBOct: BOOL;
	mxROct: BOOL;
	mxIP: BOOL;
	mxRCon: BOOL;
	mxYCon: BOOL;
	mxBCon: BOOL;
END_VAR
VAR_OUTPUT
	
END_VAR
VAR
	TASK: INT;
	qxScanBuffer_1:BOOL;
	qxScanBuffer_2:BOOL;
	qxScanBuffer_3:BOOL;
	qxScanContainer:BOOL;
	mxPlate: BOOL;
	mxCylinder: BOOL;
	mxOctagon: BOOL;
	mxPART2: BOOL;
	mxPART3: BOOL;
	mxPart1: BOOL;
	mxSLOT1: BOOL;
	mxSLOT2: BOOL;
END_VAR

CASE TASK OF
	0:
	
		MAIN.ixAutoLamp:=FALSE;
		MAIN.ixManualLamp:=FALSE;
		MAIN.qxABBErrorLamp:=FALSE;
		MAIN.qxABBExecutLamp:=FALSE;
	
		IF ABB_Control_FB.Auto_Mode.Q1 THEN
			GVL.mwStationStatus:=0;
			IF GVL.BufferProducts.Storage1.Quatity>0 THEN
				TASK:=2;
			ELSE
				TASK:=1;
			END_IF
		ELSIF ABB_Control_FB.Manual_Mode.Q1 THEN
			GVL.mwStationStatus:=400;
			TASK:=1000;
		ELSIF GVL.ixEmergencyStop THEN 
						MAIN.qxEmergySTLamp:=TRUE;
						GVL.mwStationStatus:=1000;
						TASK:=2001;
		END_IF
	
	// AUTO MODE
	
	// Buffers Scanning
	1:
		GVL.mwStationStatus:=0;
		MAIN.qxABBExecutLamp:=TRUE;
		ABB_Control_FB.qxScanBuffer_1:=TRUE;
		ABB_Control_FB.mxScan:=TRUE;
		MAIN.qsTask:='Scan buffers';
		MAIN.qsSubTask:='Scan buffer 1';
	
		IF mxEnable THEN
			IF mxRP THEN
				GVL.BufferProducts.Storage1.Component:= 'Red Plate';
				GVL.BufferProducts.Storage1.Quatity:=2;
			ELSIF mxYP THEN
				GVL.BufferProducts.Storage1.Component:= 'Yellow Plate';
				GVL.BufferProducts.Storage1.Quatity:=2;
			ELSIF mxBP THEN
				GVL.BufferProducts.Storage1.Component:='Blue Plate';
				GVL.BufferProducts.Storage1.Quatity:=2;
			ELSIF mxRCy THEN
				GVL.BufferProducts.Storage1.Component:= 'Red Cylinder';
				GVL.BufferProducts.Storage1.Quatity:=4;
			ELSIF mxYCy THEN
				GVL.BufferProducts.Storage1.Component:= 'Yellow Cylinder';
				GVL.BufferProducts.Storage1.Quatity:=4;
			ELSIF mxBCy THEN
				GVL.BufferProducts.Storage1.Component:= 'Blue Cylinder';
				GVL.BufferProducts.Storage1.Quatity:=4;
			ELSIF mxROct THEN
				GVL.BufferProducts.Storage1.Component:= 'Red Octagon';
				GVL.BufferProducts.Storage1.Quatity:=4;
			ELSIF mxYOct THEN
				GVL.BufferProducts.Storage1.Component:= 'Yellow Octagon';
				GVL.BufferProducts.Storage1.Quatity:=4;
			ELSIF mxBOct THEN
				GVL.BufferProducts.Storage1.Component:= 'Blue Octagon';
				GVL.BufferProducts.Storage1.Quatity:=4;
			ELSIF mxIP THEN
				GVL.BufferProducts.Storage1.Component:='InvalidPart';
				GVL.BufferProducts.Storage1.Quatity:=0;
			END_IF
		END_IF
		
		IF GVL.BufferProducts.Storage1.Quatity=0 OR GVL.BufferProducts.Storage2.Quatity=0 OR GVL.BufferProducts.Storage3.Quatity=0 THEN
			MAIN.ixEmptyBuffer:=TRUE;
		ELSE
			MAIN.ixEmptyBuffer:=FALSE;
		END_IF
		
		IF ABB_Control_FB.mxBuffer_1_scanned THEN
			TASK:=2;
		END_IF
		
		IF
			GVL.ixEmergencyStop THEN 
						MAIN.qxEmergySTLamp:=TRUE;
						GVL.mwStationStatus:=1000;
						TASK:=2001;
		END_IF
	
	2:
		GVL.mwStationStatus:=0;
		MAIN.qxABBExecutLamp:=TRUE;
		ABB_Control_FB.mxScan:=FALSE;
		ABB_Control_FB.qxScanBuffer_1:=FALSE;
		IF GVL.BufferProducts.Storage2.Quatity>0 THEN
			TASK:=3;
		ELSE
			TASK:=4;
		END_IF
		
	4:
		GVL.mwStationStatus:=0;
		MAIN.qxABBExecutLamp:=TRUE;
		ABB_Control_FB.mxScan:=TRUE;
		ABB_Control_FB.qxScanBuffer_2:=TRUE;
		MAIN.qsTask:='Scan buffers';
		MAIN.qsSubTask:='Scan buffer 2';
			
		IF mxEnable THEN
			IF mxRP THEN
				GVL.BufferProducts.Storage2.Component:= 'Red Plate';
				GVL.BufferProducts.Storage2.Quatity:=2;
			ELSIF mxYP THEN
				GVL.BufferProducts.Storage2.Component:= 'Yellow Plate';
				GVL.BufferProducts.Storage2.Quatity:=2;
			ELSIF mxBP THEN
				GVL.BufferProducts.Storage2.Component:='Blue Plate';
				GVL.BufferProducts.Storage2.Quatity:=2;
			ELSIF mxRCy THEN
				GVL.BufferProducts.Storage2.Component:= 'Red Cylinder';
				GVL.BufferProducts.Storage2.Quatity:=4;
			ELSIF mxYCy THEN
				GVL.BufferProducts.Storage2.Component:= 'Yellow Cylinder';
				GVL.BufferProducts.Storage2.Quatity:=4;
			ELSIF mxBCy THEN
				GVL.BufferProducts.Storage2.Component:= 'Blue Cylinder';
				GVL.BufferProducts.Storage2.Quatity:=4;
			ELSIF mxROct THEN
				GVL.BufferProducts.Storage2.Component:= 'Red Octagon';
				GVL.BufferProducts.Storage2.Quatity:=4;
			ELSIF mxYOct THEN
				GVL.BufferProducts.Storage2.Component:= 'Yellow Octagon';
				GVL.BufferProducts.Storage2.Quatity:=4;
			ELSIF mxBOct THEN
				GVL.BufferProducts.Storage2.Component:= 'Blue Octagon';
				GVL.BufferProducts.Storage2.Quatity:=4;
			ELSIF mxIP THEN
				GVL.BufferProducts.Storage2.Component:='InvalidPart';
				GVL.BufferProducts.Storage2.Quatity:=0;
			END_IF
		END_IF
		
		IF GVL.BufferProducts.Storage1.Quatity=0 OR GVL.BufferProducts.Storage2.Quatity=0 OR GVL.BufferProducts.Storage3.Quatity=0 THEN
			MAIN.ixEmptyBuffer:=TRUE;
		ELSE
			MAIN.ixEmptyBuffer:=FALSE;
		END_IF
		
		IF ABB_Control_FB.mxBuffer_2_scanned THEN
			TASK:=3;
		END_IF
		
		IF
			GVL.ixEmergencyStop THEN 
						MAIN.qxEmergySTLamp:=TRUE;
						GVL.mwStationStatus:=1000;
						TASK:=2001;
		END_IF
		
	3:
		GVL.mwStationStatus:=0;
		MAIN.qxABBExecutLamp:=TRUE;
		ABB_Control_FB.mxScan:=FALSE;
		ABB_Control_FB.qxScanBuffer_2:=FALSE;
		IF GVL.BufferProducts.Storage3.Quatity>0 THEN
			TASK:=5;
		ELSE
			TASK:=6;
		END_IF
	
	6:
		GVL.mwStationStatus:=0;
		MAIN.qxABBExecutLamp:=TRUE;
		ABB_Control_FB.mxScan:=TRUE;
		ABB_Control_FB.qxScanBuffer_3:=TRUE;
		MAIN.qsTask:='Scan buffers';
		MAIN.qsSubTask:='Scan buffer 3';
		
		IF mxEnable THEN
			IF mxRP THEN
				GVL.BufferProducts.Storage3.Component:= 'Red Plate';
				GVL.BufferProducts.Storage3.Quatity:=2;
			ELSIF mxYP THEN
				GVL.BufferProducts.Storage3.Component:= 'Yellow Plate';
				GVL.BufferProducts.Storage3.Quatity:=2;
			ELSIF mxBP THEN
				GVL.BufferProducts.Storage3.Component:='Blue Plate';
				GVL.BufferProducts.Storage3.Quatity:=2;
			ELSIF mxRCy THEN
				GVL.BufferProducts.Storage3.Component:= 'Red Cylinder';
				GVL.BufferProducts.Storage3.Quatity:=4;
			ELSIF mxYCy THEN
				GVL.BufferProducts.Storage3.Component:= 'Yellow Cylinder';
				GVL.BufferProducts.Storage3.Quatity:=4;
			ELSIF mxBCy THEN
				GVL.BufferProducts.Storage3.Component:= 'Blue Cylinder';
				GVL.BufferProducts.Storage3.Quatity:=4;
			ELSIF mxROct THEN
				GVL.BufferProducts.Storage3.Component:= 'Red Octagon';
				GVL.BufferProducts.Storage3.Quatity:=4;
			ELSIF mxYOct THEN
				GVL.BufferProducts.Storage3.Component:= 'Yellow Octagon';
				GVL.BufferProducts.Storage3.Quatity:=4;
			ELSIF mxBOct THEN
				GVL.BufferProducts.Storage3.Component:= 'Blue Octagon';
				GVL.BufferProducts.Storage3.Quatity:=4;
			ELSIF mxIP THEN
				GVL.BufferProducts.Storage3.Component:='InvalidPart';
				GVL.BufferProducts.Storage3.Quatity:=0;
			END_IF
		END_IF
		
		IF GVL.BufferProducts.Storage1.Quatity=0 OR GVL.BufferProducts.Storage2.Quatity=0 OR GVL.BufferProducts.Storage3.Quatity=0 THEN
			MAIN.ixEmptyBuffer:=TRUE;
		ELSE
			MAIN.ixEmptyBuffer:=FALSE;
		END_IF
		
		IF ABB_Control_FB.mxBuffer_3_scanned THEN
			TASK:=5;
		END_IF
		
		IF
			GVL.ixEmergencyStop THEN 
						MAIN.qxEmergySTLamp:=TRUE;
						GVL.mwStationStatus:=1000;
						TASK:=2001;
		END_IF
		
	5:
		GVL.mwStationStatus:=0;
		MAIN.qxABBExecutLamp:=TRUE;
		ABB_Control_FB.mxScan:=FALSE;
		ABB_Control_FB.qxScanBuffer_3:=FALSE;
		TASK:=7;
		
	7:
		MAIN.qxABBExecutLamp:=FALSE;
		ABB_Control_FB.ixGoTo_AGV:=FALSE;
		ABB_Control_FB.qxAssemblyDone:=FALSE;
		GVL.qxPalletPlacedinAGV:=FALSE;
		ABB_Control_FB.mxConLeave:=FALSE;
		GVL.mwStationStatus:=100;
		IF GVL.BufferProducts.Storage1.Quatity>0 AND GVL.BufferProducts.Storage2.Quatity>0 AND GVL.BufferProducts.Storage3.Quatity>0 THEN
			TASK:=8;
		ELSE
			TASK:=0;
		END_IF
	
	8: // Containers Scanning
		MAIN.qsTask:='Waiting for AGV';
		MAIN.qsSubTask:='';
		
		IF GVL.ixAGVatStation THEN
			GVL.mwStationStatus:=300;
			MAIN.qxABBExecutLamp:=TRUE;
			ABB_Control_FB.ixGoTo_AGV:=TRUE;
			ABB_Control_FB.mxScan:= TRUE;
			MAIN.qsTask:='Go to AGV Pos';
			MAIN.qsSubTask:='Pick Container';
			
			IF ABB_Control_FB.ABBPickLeaveContainerAGVPick_1.mxDone THEN
				MAIN.qsTask:='Go to Scanner';
				MAIN.qsSubTask:='Scanning Container';
			END_IF
			
			IF mxEnable THEN
				IF mxRCon THEN
					MAIN.qsContainer:='Red Container';
				ELSIF mxYCon THEN
					MAIN.qsContainer:='Yellow Container';
				ELSIF mxBCon THEN
					MAIN.qsContainer:='Blue Container';
				END_IF
				TASK:=9;
			END_IF
		END_IF
	
	9: // Parts Scanning
		IF ABB_Control_FB.mxContainerScanDone THEN
			TASK:=44;
		END_IF
		
		IF
			GVL.ixEmergencyStop THEN 
						MAIN.qxEmergySTLamp:=TRUE;
						GVL.mwStationStatus:=1000;
						TASK:=2001;
		END_IF
		
	44:
	
		ABB_Control_FB.ixGoTo_AGV:=FALSE;
		ABB_Control_FB.qxCon1:=TRUE;
		MAIN.qsTask:='Scan Products on Container';
		MAIN.qsSubTask:='Scan Plate';
		IF ABB_Control_FB.mxCon_1_ATtableScan THEN
			IF GVL.ixInductiveSensorinTool THEN
				MAIN.mxPlateAvailable:=TRUE;
				TASK:=10;
			ELSIF NOT GVL.ixInductiveSensorinTool THEN
				TASK:=100;
			END_IF
		END_IF
		
	10:
		ABB_Control_FB.mxCon_1_ATtableScan:=FALSE;
		ABB_Control_FB.qxCon1:=FALSE;
		TASK:=11;
		
	11:
		ABB_Control_FB.qxCon2:=TRUE;
		MAIN.qsTask:='Scan Products on Container';
		MAIN.qsSubTask:='Scan Cylinder';
		IF ABB_Control_FB.mxCon_2_ATtableScan THEN
			IF GVL.ixInductiveSensorinTool THEN
				MAIN.mxCylinderAvailable:=TRUE;
				TASK:=12;
			ELSIF NOT GVL.ixInductiveSensorinTool THEN
				TASK:=101;
			END_IF
		END_IF
		
	12:
		ABB_Control_FB.mxCon_2_ATtableScan:=FALSE;
		ABB_Control_FB.qxCon2:=FALSE;
		TASK:=13;
		
	13:
		ABB_Control_FB.qxCon3:=TRUE;
		MAIN.qsTask:='Scan Products on Container';
		MAIN.qsSubTask:='Scan Octagon';
		IF ABB_Control_FB.mxCon_3_ATtableScan THEN
			IF GVL.ixInductiveSensorinTool THEN
				MAIN.mxOctagonAvailable:=TRUE;
				TASK:=350;
			ELSIF NOT GVL.ixInductiveSensorinTool THEN
				TASK:=102;
			END_IF
		END_IF
		
	100:
		GVL.ixAGVatStation:=FALSE;
		ABB_Control_FB.qxCon1:=FALSE;
		
		IF MAIN.qsContainer='Red Container' THEN
			IF GVL.BufferProducts.Storage1.Component='Red Plate' AND GVL.BufferProducts.Storage1.Quatity>0 THEN
				MAIN.mwBufferID:=1;
				ABB_Control_FB.qxPart_1_Assemble:=TRUE;
				MAIN.qsTask:='Assembly';
				MAIN.qsSubTask:='Assembling Red Plate';
				GVL.BufferProducts.Storage1.Quatity:=GVL.BufferProducts.Storage1.Quatity-1;
				TASK:=200;
			ELSIF GVL.BufferProducts.Storage2.Component='Red Plate' AND GVL.BufferProducts.Storage2.Quatity>0 THEN
				MAIN.mwBufferID:=2;
				ABB_Control_FB.qxPart_2_Assemble:=TRUE;
				MAIN.qsTask:='Assembly';
				MAIN.qsSubTask:='Assembling Red Plate';
				GVL.BufferProducts.Storage2.Quatity:=GVL.BufferProducts.Storage2.Quatity-1;
				TASK:=200;
			ELSIF GVL.BufferProducts.Storage3.Component='Red Plate' AND GVL.BufferProducts.Storage3.Quatity>0 THEN
				MAIN.mwBufferID:=3;
				ABB_Control_FB.qxPart_3_Assemble:=TRUE;
				MAIN.qsTask:='Assembly';
				MAIN.qsSubTask:='Assembling Red Plate';
				GVL.BufferProducts.Storage3.Quatity:=GVL.BufferProducts.Storage3.Quatity-1;
				TASK:=200;
			ELSE
				TASK:=150;				
			END_IF
			
		ELSIF MAIN.qsContainer='Yellow Container' THEN
			IF GVL.BufferProducts.Storage1.Component='Yellow Plate' AND GVL.BufferProducts.Storage1.Quatity>0 THEN
				MAIN.mwBufferID:=1;
				ABB_Control_FB.qxPart_1_Assemble:=TRUE;
				MAIN.qsTask:='Assembly';
				MAIN.qsSubTask:='Assembling Yellow Plate';
				GVL.BufferProducts.Storage1.Quatity:=GVL.BufferProducts.Storage1.Quatity-1;
				TASK:=200;
			ELSIF GVL.BufferProducts.Storage2.Component='Yellow Plate' AND GVL.BufferProducts.Storage2.Quatity>0 THEN
				MAIN.mwBufferID:=2;
				ABB_Control_FB.qxPart_2_Assemble:=TRUE;
				MAIN.qsTask:='Assembly';
				MAIN.qsSubTask:='Assembling Yellow Plate';
				GVL.BufferProducts.Storage2.Quatity:=GVL.BufferProducts.Storage2.Quatity-1;
				TASK:=200;
			ELSIF GVL.BufferProducts.Storage3.Component='Yellow Plate' AND GVL.BufferProducts.Storage3.Quatity>0 THEN
				MAIN.mwBufferID:=3;
				ABB_Control_FB.qxPart_3_Assemble:=TRUE;
				MAIN.qsTask:='Assembly';
				MAIN.qsSubTask:='Assembling Yellow Plate';
				GVL.BufferProducts.Storage3.Quatity:=GVL.BufferProducts.Storage3.Quatity-1;
				TASK:=200;
			ELSE
				TASK:=150;
			END_IF
			
		ELSIF MAIN.qsContainer='Blue Container' THEN
			IF GVL.BufferProducts.Storage1.Component='Blue Plate' AND GVL.BufferProducts.Storage1.Quatity>0 THEN
				MAIN.mwBufferID:=1;
				ABB_Control_FB.qxPart_1_Assemble:=TRUE;
				MAIN.qsTask:='Assembly';
				MAIN.qsSubTask:='Assembling Blue Plate';
				GVL.BufferProducts.Storage1.Quatity:=GVL.BufferProducts.Storage1.Quatity-1;
				TASK:=200;
			ELSIF GVL.BufferProducts.Storage2.Component='Blue Plate' AND GVL.BufferProducts.Storage2.Quatity>0 THEN
				MAIN.mwBufferID:=2;
				ABB_Control_FB.qxPart_2_Assemble:=TRUE;
				MAIN.qsTask:='Assembly';
				MAIN.qsSubTask:='Assembling Blue Plate';
				GVL.BufferProducts.Storage2.Quatity:=GVL.BufferProducts.Storage2.Quatity-1;
				TASK:=200;
			ELSIF GVL.BufferProducts.Storage3.Component='Blue Plate' AND GVL.BufferProducts.Storage3.Quatity>0 THEN
				MAIN.mwBufferID:=3;
				ABB_Control_FB.qxPart_3_Assemble:=TRUE;
				MAIN.qsTask:='Assembly';
				MAIN.qsSubTask:='Assembling Blue Plate';
				GVL.BufferProducts.Storage3.Quatity:=GVL.BufferProducts.Storage3.Quatity-1;
				TASK:=200;
			ELSE
				TASK:=150;
			END_IF		
		END_IF
		
		IF
			GVL.ixEmergencyStop THEN 
						MAIN.qxEmergySTLamp:=TRUE;
						GVL.mwStationStatus:=1000;
						TASK:=2001;
		END_IF
	
	200:
		IF ABB_Control_FB.mxAsse_1_done THEN
			MAIN.qsTask:='Assembly';
			MAIN.qsSubTask:='Plate Assembled';
			MAIN.mxPlateAvailable:=TRUE;
			mxPlate:=TRUE;
			ABB_Control_FB.qxPart_1_Assemble:=FALSE;
			TASK:=10;
		ELSIF ABB_Control_FB.mxAsse_2_done THEN
			MAIN.qsTask:='Assembly';
			MAIN.qsSubTask:='Plate Assembled';
			MAIN.mxPlateAvailable:=TRUE;
			mxPlate:=TRUE;
			ABB_Control_FB.qxPart_2_Assemble:=FALSE;
			TASK:=10;
		ELSIF ABB_Control_FB.mxAsse_3_done THEN
			MAIN.qsTask:='Assembly';
			MAIN.qsSubTask:='Plate Assembled';
			MAIN.mxPlateAvailable:=TRUE;
			mxPlate:=TRUE;
			ABB_Control_FB.qxPart_3_Assemble:=FALSE;
			TASK:=10;
		END_IF
		
	101:
		IF MAIN.qsContainer='Red Container' THEN
			IF GVL.BufferProducts.Storage1.Component='Red Cylinder' AND GVL.BufferProducts.Storage1.Quatity>0 THEN
				MAIN.mwBufferID:=1;
				ABB_Control_FB.qxPart_1_Assemble:=TRUE;
				MAIN.qsTask:='Assembly';
				MAIN.qsSubTask:='Assembling Red Cylinder';
				GVL.BufferProducts.Storage1.Quatity:=GVL.BufferProducts.Storage1.Quatity-1;
				TASK:=201;
			ELSIF GVL.BufferProducts.Storage2.Component='Red Cylinder' AND GVL.BufferProducts.Storage2.Quatity>0 THEN
				MAIN.mwBufferID:=2;
				ABB_Control_FB.qxPart_2_Assemble:=TRUE;
				MAIN.qsTask:='Assembly';
				MAIN.qsSubTask:='Assembling Red Cylinder';
				GVL.BufferProducts.Storage2.Quatity:=GVL.BufferProducts.Storage2.Quatity-1;
				TASK:=201;
			ELSIF GVL.BufferProducts.Storage3.Component='Red Cylinder' AND GVL.BufferProducts.Storage3.Quatity>0 THEN
				MAIN.mwBufferID:=3;
				ABB_Control_FB.qxPart_3_Assemble:=TRUE;
				MAIN.qsTask:='Assembly';
				MAIN.qsSubTask:='Assembling Red Cylinder';
				GVL.BufferProducts.Storage3.Quatity:=GVL.BufferProducts.Storage3.Quatity-1;
				TASK:=201;
			ELSE
				TASK:=12;				
			END_IF
			
		ELSIF MAIN.qsContainer='Yellow Container' THEN
			IF GVL.BufferProducts.Storage1.Component='Yellow Cylinder' AND GVL.BufferProducts.Storage1.Quatity>0 THEN
				MAIN.mwBufferID:=1;
				ABB_Control_FB.qxPart_1_Assemble:=TRUE;
				MAIN.qsTask:='Assembly';
				MAIN.qsSubTask:='Assembling Yellow Cylinder';
				GVL.BufferProducts.Storage1.Quatity:=GVL.BufferProducts.Storage1.Quatity-1;
				TASK:=201;
			ELSIF GVL.BufferProducts.Storage2.Component='Yellow Cylinder' AND GVL.BufferProducts.Storage2.Quatity>0 THEN
				MAIN.mwBufferID:=2;
				ABB_Control_FB.qxPart_2_Assemble:=TRUE;
				MAIN.qsTask:='Assembly';
				MAIN.qsSubTask:='Assembling Yellow Cylinder';
				GVL.BufferProducts.Storage2.Quatity:=GVL.BufferProducts.Storage2.Quatity-1;
				TASK:=201;
			ELSIF GVL.BufferProducts.Storage3.Component='Yellow Cylinder' AND GVL.BufferProducts.Storage3.Quatity>0 THEN
				MAIN.mwBufferID:=3;
				ABB_Control_FB.qxPart_3_Assemble:=TRUE;
				MAIN.qsTask:='Assembly';
				MAIN.qsSubTask:='Assembling Yellow Cylinder';
				GVL.BufferProducts.Storage3.Quatity:=GVL.BufferProducts.Storage3.Quatity-1;
				TASK:=201;
			ELSE
				TASK:=12;
			END_IF
			
		ELSIF MAIN.qsContainer='Blue Container' THEN
			IF GVL.BufferProducts.Storage1.Component='Blue Cylinder' AND GVL.BufferProducts.Storage1.Quatity>0 THEN
				MAIN.mwBufferID:=1;
				ABB_Control_FB.qxPart_1_Assemble:=TRUE;
				MAIN.qsTask:='Assembly';
				MAIN.qsSubTask:='Assembling Blue Cylinder';
				GVL.BufferProducts.Storage1.Quatity:=GVL.BufferProducts.Storage1.Quatity-1;
				TASK:=201;
			ELSIF GVL.BufferProducts.Storage2.Component='Blue Cylinder' AND GVL.BufferProducts.Storage2.Quatity>0 THEN
				MAIN.mwBufferID:=2;
				ABB_Control_FB.qxPart_2_Assemble:=TRUE;
				MAIN.qsTask:='Assembly';
				MAIN.qsSubTask:='Assembling Blue Cylinder';
				GVL.BufferProducts.Storage2.Quatity:=GVL.BufferProducts.Storage2.Quatity-1;
				TASK:=201;
			ELSIF GVL.BufferProducts.Storage3.Component='Blue Cylinder' AND GVL.BufferProducts.Storage3.Quatity>0 THEN
				MAIN.mwBufferID:=3;
				ABB_Control_FB.qxPart_3_Assemble:=TRUE;
				MAIN.qsTask:='Assembly';
				MAIN.qsSubTask:='Assembling Blue Cylinder';
				GVL.BufferProducts.Storage3.Quatity:=GVL.BufferProducts.Storage3.Quatity-1;
				TASK:=201;
			ELSE
				TASK:=12;
			END_IF		
		END_IF
		
		IF
			GVL.ixEmergencyStop THEN 
						MAIN.qxEmergySTLamp:=TRUE;
						GVL.mwStationStatus:=1000;
						TASK:=2001;
		END_IF
		
	102:
		ABB_Control_FB.qxCon3:=FALSE;
		IF MAIN.qsContainer='Red Container' THEN
			IF GVL.BufferProducts.Storage1.Component='Red Octagon' AND GVL.BufferProducts.Storage1.Quatity>0 THEN
				MAIN.mwBufferID:=1;
				ABB_Control_FB.qxPart_1_Assemble:=TRUE;
				MAIN.qsTask:='Assembly';
				MAIN.qsSubTask:='Assembling Red Octagon';
				GVL.BufferProducts.Storage1.Quatity:=GVL.BufferProducts.Storage1.Quatity-1;
				TASK:=600;
			ELSIF GVL.BufferProducts.Storage2.Component='Red Octagon' AND GVL.BufferProducts.Storage2.Quatity>0 THEN
				MAIN.mwBufferID:=2;
				ABB_Control_FB.qxPart_2_Assemble:=TRUE;
				MAIN.qsTask:='Assembly';
				MAIN.qsSubTask:='Assembling Red Octagon';
				GVL.BufferProducts.Storage2.Quatity:=GVL.BufferProducts.Storage2.Quatity-1;
				TASK:=600;
			ELSIF GVL.BufferProducts.Storage3.Component='Red Octagon' AND GVL.BufferProducts.Storage3.Quatity>0 THEN
				MAIN.mwBufferID:=3;
				ABB_Control_FB.qxPart_3_Assemble:=TRUE;
				MAIN.qsTask:='Assembly';
				MAIN.qsSubTask:='Assembling Red Octagon';
				GVL.BufferProducts.Storage3.Quatity:=GVL.BufferProducts.Storage3.Quatity-1;
				TASK:=600;
			ELSE
				TASK:=350;				
			END_IF
			
		ELSIF MAIN.qsContainer='Yellow Container' THEN
			IF GVL.BufferProducts.Storage1.Component='Yellow Octagon' AND GVL.BufferProducts.Storage1.Quatity>0 THEN
				MAIN.mwBufferID:=1;
				ABB_Control_FB.qxPart_1_Assemble:=TRUE;
				MAIN.qsTask:='Assembly';
				MAIN.qsSubTask:='Assembling Yellow Octagon';
				GVL.BufferProducts.Storage1.Quatity:=GVL.BufferProducts.Storage1.Quatity-1;
				TASK:=600;
			ELSIF GVL.BufferProducts.Storage2.Component='Yellow Octagon' AND GVL.BufferProducts.Storage2.Quatity>0 THEN
				MAIN.mwBufferID:=2;
				ABB_Control_FB.qxPart_2_Assemble:=TRUE;
				MAIN.qsTask:='Assembly';
				MAIN.qsSubTask:='Assembling Yellow Octagon';
				GVL.BufferProducts.Storage2.Quatity:=GVL.BufferProducts.Storage2.Quatity-1;
				TASK:=600;
			ELSIF GVL.BufferProducts.Storage3.Component='Yellow Octagon' AND GVL.BufferProducts.Storage3.Quatity>0 THEN
				MAIN.mwBufferID:=3;
				ABB_Control_FB.qxPart_3_Assemble:=TRUE;
				MAIN.qsTask:='Assembly';
				MAIN.qsSubTask:='Assembling Yellow Octagon';
				GVL.BufferProducts.Storage3.Quatity:=GVL.BufferProducts.Storage3.Quatity-1;
				TASK:=600;
			ELSE
				TASK:=350;
			END_IF
			
		ELSIF MAIN.qsContainer='Blue Container' THEN
			IF GVL.BufferProducts.Storage1.Component='Blue Octagon' AND GVL.BufferProducts.Storage1.Quatity>0 THEN
				MAIN.mwBufferID:=1;
				ABB_Control_FB.qxPart_1_Assemble:=TRUE;
				MAIN.qsTask:='Assembly';
				MAIN.qsSubTask:='Assembling Blue Octagon';
				GVL.BufferProducts.Storage1.Quatity:=GVL.BufferProducts.Storage1.Quatity-1;
				TASK:=600;
			ELSIF GVL.BufferProducts.Storage2.Component='Blue Octagon' AND GVL.BufferProducts.Storage2.Quatity>0 THEN
				MAIN.mwBufferID:=2;
				ABB_Control_FB.qxPart_2_Assemble:=TRUE;
				MAIN.qsTask:='Assembly';
				MAIN.qsSubTask:='Assembling Blue Octagon';
				GVL.BufferProducts.Storage2.Quatity:=GVL.BufferProducts.Storage2.Quatity-1;
				TASK:=600;
			ELSIF GVL.BufferProducts.Storage3.Component='Blue Octagon' AND GVL.BufferProducts.Storage3.Quatity>0 THEN
				MAIN.mwBufferID:=3;
				ABB_Control_FB.qxPart_3_Assemble:=TRUE;
				MAIN.qsTask:='Assembly';
				MAIN.qsSubTask:='Assembling Blue Octagon';
				GVL.BufferProducts.Storage3.Quatity:=GVL.BufferProducts.Storage3.Quatity-1;
				TASK:=600;
			ELSE
				TASK:=350;
			END_IF		
		END_IF
		
		IF
			GVL.ixEmergencyStop THEN 
						MAIN.qxEmergySTLamp:=TRUE;
						GVL.mwStationStatus:=1000;
						TASK:=2001;
		END_IF
		
	201: 
		IF ABB_Control_FB.mxAsse_1_done THEN
			MAIN.qsTask:='Assembly';
			MAIN.qsSubTask:='Cylinder Assembled';
			MAIN.mxCylinderAvailable:=TRUE;
			ABB_Control_FB.qxPart_1_Assemble:=FALSE;
			TASK:=12;
		ELSIF ABB_Control_FB.mxAsse_2_done THEN
			MAIN.qsTask:='Assembly';
			MAIN.qsSubTask:='Cylinder Assembled';
			MAIN.mxCylinderAvailable:=TRUE;
			ABB_Control_FB.qxPart_2_Assemble:=FALSE;
			TASK:=12;
		ELSIF ABB_Control_FB.mxAsse_3_done THEN
			MAIN.qsTask:='Assembly';
			MAIN.qsSubTask:='Cylinder Assembled';
			MAIN.mxCylinderAvailable:=TRUE;
			ABB_Control_FB.qxPart_3_Assemble:=FALSE;
			TASK:=12;
		END_IF
	
	600:
		IF ABB_Control_FB.mxAsse_1_done THEN
			MAIN.qsTask:='Assembly';
			MAIN.qsSubTask:='Octagon Assembled';
			MAIN.mxOctagonAvailable:=TRUE;
			mxOctagon:=TRUE;
			ABB_Control_FB.qxPart_1_Assemble:=FALSE;
			TASK:=700;
		ELSIF ABB_Control_FB.mxAsse_2_done THEN
			MAIN.qsTask:='Assembly';
			MAIN.qsSubTask:='Octagon Assembled';
			MAIN.mxOctagonAvailable:=TRUE;
			mxOctagon:=TRUE;
			ABB_Control_FB.qxPart_2_Assemble:=FALSE;
			TASK:=700;
		ELSIF ABB_Control_FB.mxAsse_3_done THEN
			MAIN.qsTask:='Assembly';
			MAIN.qsSubTask:='Octagon Assembled';
			MAIN.mxOctagonAvailable:=TRUE;
			mxOctagon:=TRUE;
			ABB_Control_FB.qxPart_3_Assemble:=FALSE;
			TASK:=700;
		END_IF
		
	700:
		IF MAIN.mxPlateAvailable AND MAIN.mxCylinderAvailable AND MAIN.mxOctagonAvailable THEN
			ABB_Control_FB.qxAssemblyDone:=TRUE;
			GVL.qsOrderFornextAssembly:='Assembled Product';
			IF ABB_Control_FB.mxConLeave THEN
				MAIN.mxPlateAvailable:=FALSE;
				MAIN.mxCylinderAvailable:=FALSE;
				MAIN.mxOctagonAvailable:=FALSE;
				GVL.qxPalletPlacedinAGV:=TRUE;
				GVL.qsOrderFornextAssembly:='0';
				TASK:=7;
			END_IF
		END_IF
	
	150: // Order for Plates
		IF MAIN.qsContainer='Red Container' THEN
			GVL.qsOrderFornextAssembly:='Red Plate';
			TASK:=111;
		ELSIF MAIN.qsContainer='Yellow Container' THEN
			GVL.qsOrderFornextAssembly:='Yellow Plate';
			TASK:=111;
		ELSIF MAIN.qsContainer='Blue Container' THEN
			GVL.qsOrderFornextAssembly:='Blue Plate';
			TASK:=111;
		END_IF
		
	350: // Order for missing Parts
		ABB_Control_FB.qxCon3:=FALSE;
		ABB_Control_FB.qxPart_3_Assemble:=FALSE;
		
		IF mxCylinder OR MAIN.mxCylinderAvailable THEN
			mxPART2:=TRUE;
			TASK:=351;
		ELSE
			mxPART2:=FALSE;
			TASK:=351;
		END_IF
		
	351:
		IF mxOctagon OR MAIN.mxOctagonAvailable THEN
			mxPART3:=TRUE;
			TASK:=352;
		ELSE
			mxPART3:=FALSE;
			TASK:=352;
		END_IF
		
	352:
		IF MAIN.qsContainer='Red Container' THEN
			IF mxPART2 AND mxPART3 THEN
				GVL.qsOrderFornextAssembly:='Assembled Product';
				TASK:=111;
			ELSIF mxPART2 AND NOT mxPART3 THEN
				GVL.qsOrderFornextAssembly:='Red Octagon';
				TASK:=111;
			ELSIF NOT mxPART2 AND mxPART3 THEN
				GVL.qsOrderFornextAssembly:='Red Cylinder';
				TASK:=111;
			ELSIF NOT mxPART2 AND NOT mxPART3 THEN
				GVL.qsOrderFornextAssembly:='Red Cylinder';
				TASK:=111;
			END_IF
			
		ELSIF MAIN.qsContainer='Yellow Container' THEN
			IF mxPART2 AND mxPART3 THEN
				GVL.qsOrderFornextAssembly:='Assembled Product';
				TASK:=111;
			ELSIF mxPART2 AND NOT mxPART3 THEN
				GVL.qsOrderFornextAssembly:='Yellow Octagon';
				TASK:=111;
			ELSIF NOT mxPART2 AND mxPART3 THEN
				GVL.qsOrderFornextAssembly:='Yellow Cylinder';
				TASK:=111;
			ELSIF NOT mxPART2 AND NOT mxPART3 THEN
				GVL.qsOrderFornextAssembly:='Yellow Cylinder';
				TASK:=111;
			END_IF
			
		ELSIF MAIN.qsContainer='Blue Container' THEN
			IF mxPART2 AND mxPART3 THEN
				GVL.qsOrderFornextAssembly:='Assembled Product';
				TASK:=111;
			ELSIF mxPART2 AND NOT mxPART3 THEN
				GVL.qsOrderFornextAssembly:='Blue Octagon';
				TASK:=111;
			ELSIF NOT mxPART2 AND mxPART3 THEN
				GVL.qsOrderFornextAssembly:='Blue Cylinder';
				TASK:=111;
			ELSIF NOT mxPART2 AND NOT mxPART3 THEN
				GVL.qsOrderFornextAssembly:='Blue Cylinder';
				TASK:=111;
			END_IF
		END_IF
		
		
	111:
		ABB_Control_FB.qxPart_1_Assemble:=FALSE;
		ABB_Control_FB.qxPart_2_Assemble:=FALSE;
		ABB_Control_FB.qxPart_3_Assemble:=FALSE;
		ABB_Control_FB.qxCon1:=FALSE;
		ABB_Control_FB.qxCon2:=FALSE;
		ABB_Control_FB.qxCon3:=FALSE;
		ABB_Control_FB.ixGoTo_AGV:=FALSE;
		ABB_Control_FB.qxScanBuffer_1:=FALSE;
		ABB_Control_FB.qxScanBuffer_2:=FALSE;
		ABB_Control_FB.qxScanBuffer_3:=FALSE;
		mxPART2:=FALSE;
		mxPART3:=FALSE;
		ABB_Control_FB.qxAssemblyDone:=TRUE;
		GVL.qsOrderFornextAssembly:='Assembled Product';
		IF ABB_Control_FB.ABBGotoAGVPos_Assembled.mxEnable THEN
			MAIN.qsTask:='Go to AGV Pos';
			MAIN.qsSubTask:='Leave Container';
			TASK:=121;
		END_IF
		
	121:
		IF ABB_Control_FB.mxConLeave THEN
			mxPlate:=FALSE;
			mxCylinder:=FALSE;
			mxOctagon:=FALSE;
			MAIN.mxPlateAvailable:=FALSE;
			MAIN.mxCylinderAvailable:=FALSE;
			MAIN.mxOctagonAvailable:=FALSE;
			GVL.qxPalletPlacedinAGV:=TRUE;
			GVL.qsOrderFornextAssembly:='0';
			MAIN.qsContainer:='';
			TASK:=7;
		END_IF
		
		
	// MANUAL MODE
	
	1000:
		GVL.mwStationStatus:=400;
		IF ABB_Control_FB.ixGotoHome THEN
			ABB_Control_FB.qxGotoHome:=TRUE;
			MAIN.qxABBExecutLamp:=TRUE;
			TASK:=1100;
		ELSIF ABB_Control_FB.ixGotoAGV THEN
			ABB_Control_FB.qxGotoAGV:=TRUE;
			MAIN.qxABBExecutLamp:=TRUE;
			TASK:=1200;
		ELSIF ABB_Control_FB.ixGotoTable THEN
			ABB_Control_FB.qxGotoTable:=TRUE;
			MAIN.qxABBExecutLamp:=TRUE;
			TASK:=1300;
		ELSIF ABB_Control_FB.ixGotoBuffer THEN
			ABB_Control_FB.qxGotoBuffer:=TRUE;
			MAIN.qxABBExecutLamp:=TRUE;
			TASK:=1400;
		ELSIF ABB_Control_FB.ixGotoScanner THEN
			ABB_Control_FB.qxGotoScanner:=TRUE;
			MAIN.qxABBExecutLamp:=TRUE;
			TASK:=1500;
		ELSIF ABB_Control_FB.ixPickBuffer1 THEN
			ABB_Control_FB.qxPickBuffer1:=TRUE;
			MAIN.qxABBExecutLamp:=TRUE;
			TASK:=1600;
		ELSIF ABB_Control_FB.ixLeaveBuffer1 THEN
			ABB_Control_FB.qxLeaveBuffer1:=TRUE;
			MAIN.qxABBExecutLamp:=TRUE;
			TASK:=1700;
		ELSIF ABB_Control_FB.ixPickBuffer2 THEN
			ABB_Control_FB.qxPickBuffer2:=TRUE;
			MAIN.qxABBExecutLamp:=TRUE;
			TASK:=1600;
		ELSIF ABB_Control_FB.ixLeaveBuffer2 THEN
			ABB_Control_FB.qxLeaveBuffer2:=TRUE;
			MAIN.qxABBExecutLamp:=TRUE;
			TASK:=1700;
		ELSIF ABB_Control_FB.ixPickBuffer3 THEN
			ABB_Control_FB.qxPickBuffer3:=TRUE;
			MAIN.qxABBExecutLamp:=TRUE;
			TASK:=1600;
		ELSIF ABB_Control_FB.ixLeaveBuffer3 THEN
			ABB_Control_FB.qxLeaveBuffer3:=TRUE;
			MAIN.qxABBExecutLamp:=TRUE;
			TASK:=1700;
		ELSIF ABB_Control_FB.ixPickScanner THEN
			ABB_Control_FB.qxPickScanner:=TRUE;
			MAIN.qxABBExecutLamp:=TRUE;
			TASK:=1800;
		ELSIF ABB_Control_FB.ixLeaveScanner THEN
			ABB_Control_FB.qxLeaveScanner:=TRUE;
			MAIN.qxABBExecutLamp:=TRUE;
			TASK:=1900;
		ELSIF ABB_Control_FB.ixPickAGV THEN
			ABB_Control_FB.qxPickAGV:=TRUE;
			MAIN.qxABBExecutLamp:=TRUE;
			TASK:=2000;
		ELSIF ABB_Control_FB.ixLeaveAGV THEN
			ABB_Control_FB.qxLeaveAGV:=TRUE;
			MAIN.qxABBExecutLamp:=TRUE;
			TASK:=2100;
		ELSIF ABB_Control_FB.ixPickTable THEN
			ABB_Control_FB.qxPickTable:=TRUE;
			MAIN.qxABBExecutLamp:=TRUE;
			TASK:=2500;
		ELSIF ABB_Control_FB.ixLeaveTable THEN
			ABB_Control_FB.qxLeaveTable:=TRUE;
			MAIN.qxABBExecutLamp:=TRUE;
			TASK:=2600;
		ELSIF ABB_Control_FB.ixScanBuffer THEN
			ABB_Control_FB.mxScan:=TRUE;
			IF MAIN.mwBufferID=1 THEN
				TASK:=2200;
			ELSIF MAIN.mwBufferID=2 THEN
				TASK:=2300;
			ELSIF MAIN.mwBufferID=3 THEN
				TASK:=2400;
			END_IF
		ELSIF ABB_Control_FB.ixScanContainer THEN
			ABB_Control_FB.mxScan:=TRUE;
			TASK:=2700;
		ELSIF ABB_Control_FB.ixScanPart1 THEN
			MAIN.qxABBExecutLamp:=TRUE;
			TASK:=2800;
		ELSIF ABB_Control_FB.ixScanPart2 THEN
			MAIN.qxABBExecutLamp:=TRUE;
			TASK:=2900;
		ELSIF ABB_Control_FB.ixScanPart3 THEN
			MAIN.qxABBExecutLamp:=TRUE;
			TASK:=3000;
		ELSIF ABB_Control_FB.ixAssemble1 THEN
			MAIN.qxABBExecutLamp:=TRUE;
			GVL.BufferProducts.Storage1.Quatity:=GVL.BufferProducts.Storage1.Quatity-1;
			TASK:=3100;
		ELSIF ABB_Control_FB.ixAssemble2 THEN
			MAIN.qxABBExecutLamp:=TRUE;
			GVL.BufferProducts.Storage2.Quatity:=GVL.BufferProducts.Storage2.Quatity-1;
			TASK:=3200;
		ELSIF ABB_Control_FB.ixAssemble3 THEN
			MAIN.qxABBExecutLamp:=TRUE;
			GVL.BufferProducts.Storage3.Quatity:=GVL.BufferProducts.Storage3.Quatity-1;
			TASK:=3300;
		ELSIF ABB_Control_FB.ixSendOrder THEN
			TASK:=3400;
		ELSIF ABB_Control_FB.ixFinishOrder THEN
			TASK:=3900;
			
		END_IF
		
	1100:
		IF ABB_Control_FB.qxHOME THEN
			MAIN.qxABBExecutLamp:=FALSE;
			ABB_Control_FB.qxGotoHome:=FALSE;
			ABB_Control_FB.ixGotoHome:=FALSE;
			TASK:=1000;
		END_IF
		
	1200:
		IF ABB_Control_FB.qxAGV THEN
			MAIN.qxABBExecutLamp:=FALSE;
			ABB_Control_FB.qxGotoAGV:=FALSE;
			ABB_Control_FB.ixGotoAGV:=FALSE;
			TASK:=1000;
		END_IF
		
	1300:
		IF ABB_Control_FB.qxTABLE THEN
			MAIN.qxABBExecutLamp:=FALSE;
			ABB_Control_FB.qxGotoTable:=FALSE;
			ABB_Control_FB.ixGotoTable:=FALSE;
			TASK:=1000;
		END_IF
		
	1400:
		IF ABB_Control_FB.qxBUFFER THEN
			MAIN.qxABBExecutLamp:=FALSE;
			ABB_Control_FB.qxGotoBuffer:=FALSE;
			ABB_Control_FB.ixGotoBuffer:=FALSE;
			TASK:=1000;
		END_IF
		
	1500:
		IF ABB_Control_FB.qxSCANNER THEN
			MAIN.qxABBExecutLamp:=FALSE;
			ABB_Control_FB.qxGotoScanner:=FALSE;
			ABB_Control_FB.ixGotoScanner:=FALSE;
			TASK:=1000;
		END_IF
		
	1600:
		IF ABB_Control_FB.qxBufferPicked1 THEN
			MAIN.qxABBExecutLamp:=FALSE;
			ABB_Control_FB.qxPickBuffer1:=FALSE;
			ABB_Control_FB.ixPickBuffer1:=FALSE;
			ABB_Control_FB.qxPickBuffer2:=FALSE;
			ABB_Control_FB.ixPickBuffer2:=FALSE;
			ABB_Control_FB.qxPickBuffer3:=FALSE;
			ABB_Control_FB.ixPickBuffer3:=FALSE;
			TASK:=1000;
		END_IF
		
	1700:
		IF ABB_Control_FB.qxBufferLeft1 THEN
			MAIN.qxABBExecutLamp:=FALSE;
			ABB_Control_FB.qxPickBuffer1:=FALSE;
			ABB_Control_FB.ixPickBuffer1:=FALSE;
			ABB_Control_FB.qxPickBuffer2:=FALSE;
			ABB_Control_FB.ixPickBuffer2:=FALSE;
			ABB_Control_FB.qxPickBuffer3:=FALSE;
			ABB_Control_FB.ixPickBuffer3:=FALSE;
			TASK:=1000;
		END_IF
		
	1800:
		IF ABB_Control_FB.qxPickedScanner THEN
			MAIN.qxABBExecutLamp:=FALSE;
			ABB_Control_FB.qxPickScanner:=FALSE;
			ABB_Control_FB.ixPickScanner:=FALSE;
			TASK:=1000;
		END_IF
		
	1900:
		IF ABB_Control_FB.qxLeftScanner THEN
			MAIN.qxABBExecutLamp:=FALSE;
			ABB_Control_FB.qxLeaveScanner:=FALSE;
			ABB_Control_FB.ixLeaveScanner:=FALSE;
			TASK:=1000;
		END_IF
		
	2000:
		IF ABB_Control_FB.qxPickedAGV THEN
			MAIN.qxABBExecutLamp:=FALSE;
			GVL.qxPickedfromAGV:=TRUE;
			ABB_Control_FB.qxPickAGV:=FALSE;
			ABB_Control_FB.ixPickAGV:=FALSE;
			TASK:=1000;
		END_IF
		
	2100:
		IF ABB_Control_FB.qxLeftAGV THEN
			MAIN.qxABBExecutLamp:=FALSE;
			GVL.qxPalletPlacedinAGV:=TRUE;
			ABB_Control_FB.qxLeaveAGV:=FALSE;
			ABB_Control_FB.ixLeaveAGV:=FALSE;
			TASK:=1000;
		END_IF
		
	2200:
			IF mxRP THEN
				GVL.BufferProducts.Storage1.Component:= 'Red Plate';
				GVL.BufferProducts.Storage1.Quatity:=2;
			ELSIF mxYP THEN
				GVL.BufferProducts.Storage1.Component:= 'Yellow Plate';
				GVL.BufferProducts.Storage1.Quatity:=2;
			ELSIF mxBP THEN
				GVL.BufferProducts.Storage1.Component:='Blue Plate';
				GVL.BufferProducts.Storage1.Quatity:=2;
			ELSIF mxRCy THEN
				GVL.BufferProducts.Storage1.Component:= 'Red Cylinder';
				GVL.BufferProducts.Storage1.Quatity:=4;
			ELSIF mxYCy THEN
				GVL.BufferProducts.Storage1.Component:= 'Yellow Cylinder';
				GVL.BufferProducts.Storage1.Quatity:=4;
			ELSIF mxBCy THEN
				GVL.BufferProducts.Storage1.Component:= 'Blue Cylinder';
				GVL.BufferProducts.Storage1.Quatity:=4;
			ELSIF mxROct THEN
				GVL.BufferProducts.Storage1.Component:= 'Red Octagon';
				GVL.BufferProducts.Storage1.Quatity:=4;
			ELSIF mxYOct THEN
				GVL.BufferProducts.Storage1.Component:= 'Yellow Octagon';
				GVL.BufferProducts.Storage1.Quatity:=4;
			ELSIF mxBOct THEN
				GVL.BufferProducts.Storage1.Component:= 'Blue Octagon';
				GVL.BufferProducts.Storage1.Quatity:=4;
			ELSIF mxIP THEN
				GVL.BufferProducts.Storage1.Component:='InvalidPart';
				GVL.BufferProducts.Storage1.Quatity:=0;
			END_IF
			TASK:=1000;
			
	2300:
			IF mxRP THEN
				GVL.BufferProducts.Storage1.Component:= 'Red Plate';
				GVL.BufferProducts.Storage1.Quatity:=2;
			ELSIF mxYP THEN
				GVL.BufferProducts.Storage1.Component:= 'Yellow Plate';
				GVL.BufferProducts.Storage1.Quatity:=2;
			ELSIF mxBP THEN
				GVL.BufferProducts.Storage1.Component:='Blue Plate';
				GVL.BufferProducts.Storage1.Quatity:=2;
			ELSIF mxRCy THEN
				GVL.BufferProducts.Storage1.Component:= 'Red Cylinder';
				GVL.BufferProducts.Storage1.Quatity:=4;
			ELSIF mxYCy THEN
				GVL.BufferProducts.Storage1.Component:= 'Yellow Cylinder';
				GVL.BufferProducts.Storage1.Quatity:=4;
			ELSIF mxBCy THEN
				GVL.BufferProducts.Storage1.Component:= 'Blue Cylinder';
				GVL.BufferProducts.Storage1.Quatity:=4;
			ELSIF mxROct THEN
				GVL.BufferProducts.Storage1.Component:= 'Red Octagon';
				GVL.BufferProducts.Storage1.Quatity:=4;
			ELSIF mxYOct THEN
				GVL.BufferProducts.Storage1.Component:= 'Yellow Octagon';
				GVL.BufferProducts.Storage1.Quatity:=4;
			ELSIF mxBOct THEN
				GVL.BufferProducts.Storage1.Component:= 'Blue Octagon';
				GVL.BufferProducts.Storage1.Quatity:=4;
			ELSIF mxIP THEN
				GVL.BufferProducts.Storage1.Component:='InvalidPart';
				GVL.BufferProducts.Storage1.Quatity:=0;
			END_IF
			TASK:=1000;
			
	2400:
			IF mxRP THEN
				GVL.BufferProducts.Storage1.Component:= 'Red Plate';
				GVL.BufferProducts.Storage1.Quatity:=2;
			ELSIF mxYP THEN
				GVL.BufferProducts.Storage1.Component:= 'Yellow Plate';
				GVL.BufferProducts.Storage1.Quatity:=2;
			ELSIF mxBP THEN
				GVL.BufferProducts.Storage1.Component:='Blue Plate';
				GVL.BufferProducts.Storage1.Quatity:=2;
			ELSIF mxRCy THEN
				GVL.BufferProducts.Storage1.Component:= 'Red Cylinder';
				GVL.BufferProducts.Storage1.Quatity:=4;
			ELSIF mxYCy THEN
				GVL.BufferProducts.Storage1.Component:= 'Yellow Cylinder';
				GVL.BufferProducts.Storage1.Quatity:=4;
			ELSIF mxBCy THEN
				GVL.BufferProducts.Storage1.Component:= 'Blue Cylinder';
				GVL.BufferProducts.Storage1.Quatity:=4;
			ELSIF mxROct THEN
				GVL.BufferProducts.Storage1.Component:= 'Red Octagon';
				GVL.BufferProducts.Storage1.Quatity:=4;
			ELSIF mxYOct THEN
				GVL.BufferProducts.Storage1.Component:= 'Yellow Octagon';
				GVL.BufferProducts.Storage1.Quatity:=4;
			ELSIF mxBOct THEN
				GVL.BufferProducts.Storage1.Component:= 'Blue Octagon';
				GVL.BufferProducts.Storage1.Quatity:=4;
			ELSIF mxIP THEN
				GVL.BufferProducts.Storage1.Component:='InvalidPart';
				GVL.BufferProducts.Storage1.Quatity:=0;
			END_IF
			TASK:=1000;
			
	2500:
		IF ABB_Control_FB.qxPickedTable THEN
			MAIN.qxABBExecutLamp:=FALSE;
			ABB_Control_FB.qxPickTable:=FALSE;
			ABB_Control_FB.ixPickTable:=FALSE;
			TASK:=1000;
		END_IF
		
	2600:
		IF ABB_Control_FB.qxLeftTable THEN
			MAIN.qxABBExecutLamp:=FALSE;
			ABB_Control_FB.qxLeaveTable:=FALSE;
			ABB_Control_FB.ixLeaveTable:=FALSE;
			TASK:=1000;
		END_IF
		
	2700:
				IF mxRCon THEN
					MAIN.qsContainer:='Red Container';
				ELSIF mxYCon THEN
					MAIN.qsContainer:='Yellow Container';
				ELSIF mxBCon THEN
					MAIN.qsContainer:='Blue Container';
				END_IF
				TASK:=1000;
				
	2800:
		IF ABB_Control_FB.mxCon_1_ATtableScan THEN
			IF GVL.ixInductiveSensorinTool THEN
				MAIN.mxPlateAvailable:=TRUE;
				TASK:=1000;
				ABB_Control_FB.ixScanPart1:=FALSE;
				MAIN.qxABBExecutLamp:=FALSE;
			ELSIF NOT GVL.ixInductiveSensorinTool THEN
				ABB_Control_FB.ixScanPart1:=FALSE;
				MAIN.qxABBExecutLamp:=FALSE;
				TASK:=1000;
			END_IF
		END_IF
		
	2900:
		IF ABB_Control_FB.mxCon_2_ATtableScan THEN
			IF GVL.ixInductiveSensorinTool THEN
				MAIN.mxCylinderAvailable:=TRUE;
				TASK:=1000;
				ABB_Control_FB.ixScanPart2:=FALSE;
				MAIN.qxABBExecutLamp:=FALSE;
			ELSIF NOT GVL.ixInductiveSensorinTool THEN
				ABB_Control_FB.ixScanPart2:=FALSE;
				MAIN.qxABBExecutLamp:=FALSE;
				TASK:=1000;
			END_IF
		END_IF
		
	3000:
		IF ABB_Control_FB.mxCon_2_ATtableScan THEN
			IF GVL.ixInductiveSensorinTool THEN
				MAIN.mxOctagonAvailable:=TRUE;
				TASK:=1000;
				ABB_Control_FB.ixScanPart3:=FALSE;
				MAIN.qxABBExecutLamp:=FALSE;
			ELSIF NOT GVL.ixInductiveSensorinTool THEN
				ABB_Control_FB.ixScanPart3:=FALSE;
				MAIN.qxABBExecutLamp:=FALSE;
				TASK:=1000;
			END_IF
		END_IF
		
	3100:
		IF ABB_Control_FB.mxAsse_1_done THEN
			mxPart1:=TRUE;
			ABB_Control_FB.ixAssemble1:=FALSE;
			MAIN.qxABBExecutLamp:=FALSE;
			TASK:=1000;
		END_IF
		
	3200:
		IF ABB_Control_FB.mxAsse_2_done THEN
			mxPart2:=TRUE;
			ABB_Control_FB.ixAssemble2:=FALSE;
			MAIN.qxABBExecutLamp:=FALSE;
			TASK:=1000;
		END_IF
		
	3300:
		IF ABB_Control_FB.mxAsse_3_done THEN
			mxPart3:=TRUE;
			ABB_Control_FB.ixAssemble3:=FALSE;
			MAIN.qxABBExecutLamp:=FALSE;
			TASK:=1000;
		END_IF
		
	3400:
		IF NOT MAIN.mxPlateAvailable AND mxPart1 THEN
			IF MAIN.qsContainer='Red Container' THEN
				GVL.qsOrderFornextAssembly:='Red Plate';
			ELSIF MAIN.qsContainer='Yellow Container' THEN
				GVL.qsOrderFornextAssembly:='Yellow Plate';
			ELSIF MAIN.qsContainer='Blue Container' THEN
				GVL.qsOrderFornextAssembly:='Blue Plate';
			ELSE
				TASK:=3500;
			END_IF
		END_IF
		
	3500:
		IF mxPart2 OR MAIN.mxCylinderAvailable THEN
			mxSLOT1:=TRUE;
			TASK:=3600;
		ELSE
			mxSLOT1:=FALSE;
			TASK:=3600;
		END_IF
		
	3600:
	 	IF mxPART3 OR MAIN.mxOctagonAvailable THEN
		 	mxSLOT2:=TRUE;
		 	TASK:=3800;
		ELSE
			mxSLOT2:=FALSE;
			TASK:=3800;
	 	END_IF
	 
	3800:
		IF MAIN.qsContainer='Yellow Container' THEN
			IF mxSLOT1 AND mxSLOT2 THEN 
					   gvl.qsOrderFornextAssembly:='Assembled Product';
					   TASK:=3900;
					   ELSIF mxSLOT1 AND NOT mxSLOT2 THEN 
						   gvl.qsOrderFornextAssembly:='Yellow Octagon';
					    TASK:=3900;
					   ELSIF NOT mxSLOT1 AND mxSLOT2 THEN 
						   gvl.qsOrderFornextAssembly:='Yellow Cylinder';
					    TASk:=3900;
					   ELSIF NOT mxSLOT1 AND NOT mxSLOT2 THEN
						  gvl.qsOrderFornextAssembly:='Yellow Cylinder';
					    TASK:=3900; 
				   END_IF
				   
		ELSIF MAIN.qsContainer='Red Container' THEN
			IF mxSLOT1 AND mxSLOT2 THEN 
					   gvl.qsOrderFornextAssembly:='Assembled Product';
					   TASK:=3900;
					   ELSIF mxSLOT1 AND NOT mxSLOT2 THEN 
						   gvl.qsOrderFornextAssembly:='Red Octagon';
					    TASK:=3900;
					   ELSIF NOT mxSLOT1 AND mxSLOT2 THEN 
						   gvl.qsOrderFornextAssembly:='Red Cylinder';
					    TASk:=3900;
					   ELSIF NOT mxSLOT1 AND NOT mxSLOT2 THEN
						  gvl.qsOrderFornextAssembly:='Red Cylinder';
					    TASK:=3900; 
				   END_IF
				   
		ELSIF MAIN.qsContainer='Blue Container' THEN
			IF mxSLOT1 AND mxSLOT2 THEN 
					   gvl.qsOrderFornextAssembly:='Assembled Product';
					   TASK:=3900;
					   ELSIF mxSLOT1 AND NOT mxSLOT2 THEN 
						   gvl.qsOrderFornextAssembly:='Blue Octagon';
					    TASK:=3900;
					   ELSIF NOT mxSLOT1 AND mxSLOT2 THEN 
						   gvl.qsOrderFornextAssembly:='Blue Cylinder';
					    TASk:=3900;
					   ELSIF NOT mxSLOT1 AND NOT mxSLOT2 THEN
						  gvl.qsOrderFornextAssembly:='Blue Cylinder';
					    TASK:=3900; 
				   END_IF
		
		END_IF
		
	3900:
		IF ABB_Control_FB.ixFinishOrder THEN
			ABB_Control_FB.mxAsse_1_done:=FALSE;
			ABB_Control_FB.mxAsse_2_done:=FALSE;
			ABB_Control_FB.mxAsse_3_done:=FALSE;
			GVL.qsOrderFornextAssembly:='0';
			TASK:=1000;
		END_IF
		
	2001: // Emergency Stop
		ABB_Control_FB.qxScanBuffer_1:=FALSE;
		ABB_Control_FB.qxScanBuffer_2:=FALSE;
		ABB_Control_FB.qxScanBuffer_3:=FALSE;
		ABB_Control_FB.ixGoTo_AGV:=FALSE;
		ABB_Control_FB.qxCon1:=FALSE;
		ABB_Control_FB.qxCon2:=FALSE;
		ABB_Control_FB.qxCon3:=FALSE;
		ABB_Control_FB.qxPart_1_Assemble:=FALSE;
		ABB_Control_FB.qxPart_2_Assemble:=FALSE;
		ABB_Control_FB.qxPart_3_Assemble:=FALSE;
		ABB_Control_FB.qxAssemblyDone:=FALSE;
	 
	
END_CASE

END_FUNCTION_BLOCK

// ---- POUs/Sensor_Sense.TcPOU
FUNCTION_BLOCK Sensor_Sense
VAR_INPUT
	mxEnable: BOOL;
END_VAR
VAR_OUTPUT
	Product:STRING;
	mxINVALIDPRODUCT:BOOL;
	mxREDPLATE:BOOL;
	mxYELLOWPLATE:BOOL;
	mxBLUEPLATE:BOOL;
	mxREDCYLINDER:BOOL;
	mxYELLOWCYLINDER:BOOL;
	mxBLUECYLINDER:BOOL;
	mxREDOCTAGON:BOOL;
	mxYELLOWOCTAGON:BOOL;
	mxBLUEOCTAGON:BOOL;
	mxREDCONTAINER:BOOL;
	mxYELLOWCONTAINER:BOOL;
	mxBLUECONTAINER:BOOL;
END_VAR
VAR
	Sensor_Sense:BYTE;
END_VAR

IF mxEnable THEN
	Sensor_Sense.1:=gvl.ixInductiveSensor1;
	Sensor_Sense.2:=gvl.ixInductiveSensor2;
	Sensor_Sense.3:=gvl.ixInductiveSensor3;
	Sensor_Sense.4:=gvl.ixInductiveSensor4;
END_IF

IF Sensor_Sense = 0 OR Sensor_Sense = 4 OR Sensor_Sense = 2 OR Sensor_Sense = 6 THEN
 	Product:='InvalidPart';
	mxINVALIDPRODUCT:=FALSE;
END_IF

IF Sensor_Sense=16 THEN
	Product:='Blue Container';
	mxREDPLATE:=FALSE;
	mxYELLOWPLATE:=FALSE;
	mxBLUEPLATE:=FALSE;
	mxREDCYLINDER:=FALSE;
	mxYELLOWCYLINDER:=FALSE;
	mxBLUECYLINDER:=FALSE;
	mxREDOCTAGON:=FALSE;
	mxYELLOWOCTAGON:=FALSE;
	mxBLUEOCTAGON:=FALSE;
	mxREDCONTAINER:=FALSE;
	mxYELLOWCONTAINER:=FALSE;
	mxBLUECONTAINER:=TRUE;
	
END_IF

IF Sensor_Sense=8 THEN
	Product:='Yellow Container';
	mxREDPLATE:=FALSE;
	mxYELLOWPLATE:=FALSE;
	mxBLUEPLATE:=FALSE;
	mxREDCYLINDER:=FALSE;
	mxYELLOWCYLINDER:=FALSE;
	mxBLUECYLINDER:=FALSE;
	mxREDOCTAGON:=FALSE;
	mxYELLOWOCTAGON:=FALSE;
	mxBLUEOCTAGON:=FALSE;
	mxREDCONTAINER:=FALSE;
	mxYELLOWCONTAINER:=TRUE;
	mxBLUECONTAINER:=FALSE;
END_IF

IF Sensor_Sense=24 THEN
	Product:='Red Container';
	mxREDPLATE:=FALSE;
	mxYELLOWPLATE:=FALSE;
	mxBLUEPLATE:=FALSE;
	mxREDCYLINDER:=FALSE;
	mxYELLOWCYLINDER:=FALSE;
	mxBLUECYLINDER:=FALSE;
	mxREDOCTAGON:=FALSE;
	mxYELLOWOCTAGON:=FALSE;
	mxBLUEOCTAGON:=FALSE;
	mxREDCONTAINER:=TRUE;
	mxYELLOWCONTAINER:=FALSE;
	mxBLUECONTAINER:=FALSE;
END_IF

IF Sensor_Sense=20 THEN
	Product:='Blue Cylinder';
	mxREDPLATE:=FALSE;
	mxYELLOWPLATE:=FALSE;
	mxBLUEPLATE:=FALSE;
	mxREDCYLINDER:=FALSE;
	mxYELLOWCYLINDER:=FALSE;
	mxBLUECYLINDER:=TRUE;
	mxREDOCTAGON:=FALSE;
	mxYELLOWOCTAGON:=FALSE;
	mxBLUEOCTAGON:=FALSE;
	mxREDCONTAINER:=FALSE;
	mxYELLOWCONTAINER:=FALSE;
	mxBLUECONTAINER:=FALSE;
END_IF

IF Sensor_Sense=12 THEN
	Product:='Blue Octagon';
	mxREDPLATE:=FALSE;
	mxYELLOWPLATE:=FALSE;
	mxBLUEPLATE:=FALSE;
	mxREDCYLINDER:=FALSE;
	mxYELLOWCYLINDER:=FALSE;
	mxBLUECYLINDER:=FALSE;
	mxREDOCTAGON:=FALSE;
	mxYELLOWOCTAGON:=FALSE;
	mxBLUEOCTAGON:=TRUE;
	mxREDCONTAINER:=FALSE;
	mxYELLOWCONTAINER:=FALSE;
	mxBLUECONTAINER:=FALSE;
END_IF

IF Sensor_Sense=28 THEN
	Product:='Blue Plate';
	mxREDPLATE:=FALSE;
	mxYELLOWPLATE:=FALSE;
	mxBLUEPLATE:=TRUE;
	mxREDCYLINDER:=FALSE;
	mxYELLOWCYLINDER:=FALSE;
	mxBLUECYLINDER:=FALSE;
	mxREDOCTAGON:=FALSE;
	mxYELLOWOCTAGON:=FALSE;
	mxBLUEOCTAGON:=FALSE;
	mxREDCONTAINER:=FALSE;
	mxYELLOWCONTAINER:=FALSE;
	mxBLUECONTAINER:=FALSE;
END_IF

IF Sensor_Sense=18 THEN
	Product:='Yellow Cylinder';
	mxREDPLATE:=FALSE;
	mxYELLOWPLATE:=FALSE;
	mxBLUEPLATE:=FALSE;
	mxREDCYLINDER:=FALSE;
	mxYELLOWCYLINDER:=TRUE;
	mxBLUECYLINDER:=FALSE;
	mxREDOCTAGON:=FALSE;
	mxYELLOWOCTAGON:=FALSE;
	mxBLUEOCTAGON:=FALSE;
	mxREDCONTAINER:=FALSE;
	mxYELLOWCONTAINER:=FALSE;
	mxBLUECONTAINER:=FALSE;
END_IF

IF Sensor_Sense=10 THEN
	Product:='Yellow Octagon';
	mxREDPLATE:=FALSE;
	mxYELLOWPLATE:=FALSE;
	mxBLUEPLATE:=FALSE;
	mxREDCYLINDER:=FALSE;
	mxYELLOWCYLINDER:=FALSE;
	mxBLUECYLINDER:=FALSE;
	mxREDOCTAGON:=FALSE;
	mxYELLOWOCTAGON:=TRUE;
	mxBLUEOCTAGON:=FALSE;
	mxREDCONTAINER:=FALSE;
	mxYELLOWCONTAINER:=FALSE;
	mxBLUECONTAINER:=FALSE;
END_IF

IF Sensor_Sense=26 THEN
	Product:='Yellow Plate';
	mxREDPLATE:=FALSE;
	mxYELLOWPLATE:=TRUE;
	mxBLUEPLATE:=FALSE;
	mxREDCYLINDER:=FALSE;
	mxYELLOWCYLINDER:=FALSE;
	mxBLUECYLINDER:=FALSE;
	mxREDOCTAGON:=FALSE;
	mxYELLOWOCTAGON:=FALSE;
	mxBLUEOCTAGON:=FALSE;
	mxREDCONTAINER:=FALSE;
	mxYELLOWCONTAINER:=FALSE;
	mxBLUECONTAINER:=FALSE;
END_IF

IF Sensor_Sense=22 THEN
	Product:='Red Cylinder';
	mxREDPLATE:=FALSE;
	mxYELLOWPLATE:=FALSE;
	mxBLUEPLATE:=FALSE;
	mxREDCYLINDER:=TRUE;
	mxYELLOWCYLINDER:=FALSE;
	mxBLUECYLINDER:=FALSE;
	mxREDOCTAGON:=FALSE;
	mxYELLOWOCTAGON:=FALSE;
	mxBLUEOCTAGON:=FALSE;
	mxREDCONTAINER:=FALSE;
	mxYELLOWCONTAINER:=FALSE;
	mxBLUECONTAINER:=FALSE;
END_IF

IF Sensor_Sense=14 THEN
	Product:='Red Octagon';
	mxREDPLATE:=FALSE;
	mxYELLOWPLATE:=FALSE;
	mxBLUEPLATE:=FALSE;
	mxREDCYLINDER:=FALSE;
	mxYELLOWCYLINDER:=FALSE;
	mxBLUECYLINDER:=FALSE;
	mxREDOCTAGON:=TRUE;
	mxYELLOWOCTAGON:=FALSE;
	mxBLUEOCTAGON:=FALSE;
	mxREDCONTAINER:=FALSE;
	mxYELLOWCONTAINER:=FALSE;
	mxBLUECONTAINER:=FALSE;
END_IF

IF Sensor_Sense=30 THEN
	Product:='Red Plate';
	mxREDPLATE:=TRUE;
	mxYELLOWPLATE:=FALSE;
	mxBLUEPLATE:=FALSE;
	mxREDCYLINDER:=FALSE;
	mxYELLOWCYLINDER:=FALSE;
	mxBLUECYLINDER:=FALSE;
	mxREDOCTAGON:=FALSE;
	mxYELLOWOCTAGON:=FALSE;
	mxBLUEOCTAGON:=FALSE;
	mxREDCONTAINER:=FALSE;
	mxYELLOWCONTAINER:=FALSE;
	mxBLUECONTAINER:=FALSE;
END_IF

END_FUNCTION_BLOCK

// ---- ABBControl/ABBGotoAGVPos.TcPOU
FUNCTION_BLOCK ABBGotoAGVPos
VAR_INPUT
	mxEnable: BOOL;
END_VAR
VAR_OUTPUT
	mxDone:BOOL;
	mxExecuting: BOOL;
	mxError: BOOL;
END_VAR
VAR
	ABB: INT;
END_VAR

